// Render the set header as a JSON object. The timestamp is emitted as the
// §2.7 clock's seconds value rather than a formatted date: a set document is
// machine input, and a numeric instant cannot be misread by a reader in another
// locale. TimeSynchronized travels with it, so a consumer can tell a trustworthy
// instant from one stamped while the clock had lost its source.
METHOD M_Header : STRING(480)
VAR_INPUT
    Info : ST_ConfigSetInfo;
END_VAR
VAR
    nameText  : STRING(480);
    rootText  : STRING(480);
    modelText : STRING(480);
    line      : STRING(480);
    used      : INT;
    ok        : BOOL;
END_VAR
M_Header := '';
IF Info.SetName = '' THEN
    RETURN;
END_IF
nameText := _M_Escape(Text := Info.SetName, Ok => ok);
IF NOT ok THEN
    RETURN;
END_IF
rootText := _M_Escape(Text := Info.RootIdentity, Ok => ok);
IF NOT ok THEN
    RETURN;
END_IF
modelText := _M_Escape(Text := Info.ModelCode, Ok => ok);
IF NOT ok THEN
    RETURN;
END_IF
line := '';
used := 0;
ok := _M_PutText(Text := '{"set":"', Line := line, Used := used)
    AND_THEN _M_Put(pText := ADR(nameText), Line := line, Used := used)
    AND_THEN _M_PutText(Text := '","root":"', Line := line, Used := used)
    AND_THEN _M_Put(pText := ADR(rootText), Line := line, Used := used)
    AND_THEN _M_PutText(Text := '","schema":', Line := line, Used := used)
    AND_THEN _M_PutText(Text := UINT_TO_STRING(Info.SetSchema), Line := line, Used := used)
    AND_THEN _M_PutText(Text := ',"configRev":', Line := line, Used := used)
    AND_THEN _M_PutText(Text := UDINT_TO_STRING(Info.ConfigRev), Line := line, Used := used)
    AND_THEN _M_PutText(Text := ',"kind":', Line := line, Used := used)
    AND_THEN _M_PutText(Text := DINT_TO_STRING(TO_DINT(Info.Kind)), Line := line, Used := used)
    AND_THEN _M_PutText(Text := ',"model":"', Line := line, Used := used)
    AND_THEN _M_Put(pText := ADR(modelText), Line := line, Used := used)
    AND_THEN _M_PutText(Text := '","records":', Line := line, Used := used)
    AND_THEN _M_PutText(Text := INT_TO_STRING(Info.RecordCount), Line := line, Used := used)
    AND_THEN _M_PutText(Text := ',"created":', Line := line, Used := used)
    AND_THEN _M_PutText(Text := UDINT_TO_STRING(DT_TO_UDINT(Info.CreatedAt)), Line := line, Used := used)
    AND_THEN _M_PutText(Text := ',"clock":', Line := line, Used := used);
IF ok THEN
    IF Info.TimeSynchronized THEN
        ok := _M_PutText(Text := '1}', Line := line, Used := used);
    ELSE
        ok := _M_PutText(Text := '0}', Line := line, Used := used);
    END_IF
END_IF
IF ok THEN
    M_Header := line;
END_IF
END_METHOD

// Read one field out of a flat JSON object line. Deliberately NOT a general
// JSON parser: the accepted shape is exactly what M_Record and M_Header emit -
// a single object of scalar members, no nesting, no arrays. Anything else is
// refused rather than half-understood, which is the §14 rule for untrusted
// input applied to a format instead of to a value.
METHOD PRIVATE _M_Field : BOOL
VAR_INPUT
    Line : STRING(480);
    Name : STRING(32);
END_VAR
VAR_OUTPUT
    Value : STRING(255);
END_VAR
VAR
    pIn   : POINTER TO BYTE;
    pOut  : POINTER TO BYTE;
    buf   : STRING(255);
    token : STRING(40);
    pTok  : POINTER TO BYTE;
    tokLen : INT;
    found : INT;
    i     : INT;
    j     : INT;
    k     : INT;
    n     : INT;
    ch    : BYTE;
    quoted : BOOL;
END_VAR
_M_Field := FALSE;
Value := '';
buf := '';
token := CONCAT('"', CONCAT(Name, '":'));   // short: CONCAT is exact here
pIn := ADR(Line);
pTok := ADR(token);
n := _M_Length(pText := pIn);               // FIND/LEN would see only 255 of it
tokLen := TO_INT(LEN(token));
found := -1;
FOR i := 0 TO n - tokLen DO
    k := 0;
    WHILE (k < tokLen) AND_THEN (pIn[i + k] = pTok[k]) DO
        k := k + 1;
    END_WHILE
    IF k = tokLen THEN
        found := i;
        EXIT;
    END_IF
END_FOR
IF found < 0 THEN
    RETURN;                                // absent: the caller decides if that is fatal
END_IF
i := found + tokLen;                          // 0-based index of the first value byte
IF i >= n THEN
    RETURN;
END_IF
pOut := ADR(buf);
j := 0;
quoted := (pIn[i] = 16#22);
IF quoted THEN
    i := i + 1;
END_IF
WHILE i < n DO
    ch := pIn[i];
    IF quoted THEN
        IF ch = 16#22 THEN
            EXIT;                          // closing quote
        END_IF
        IF ch = 16#5C THEN
            i := i + 1;                    // unescape: the next byte is literal
            IF i >= n THEN
                RETURN;                    // trailing escape: malformed, refuse
            END_IF
            ch := pIn[i];
        END_IF
    ELSE
        IF (ch = 16#2C) OR (ch = 16#7D) THEN
            EXIT;                          // ',' or '}' ends a bare number
        END_IF
    END_IF
    IF j >= 254 THEN
        RETURN;                            // longer than any value we can store
    END_IF
    pOut[j] := ch;
    j := j + 1;
    i := i + 1;
END_WHILE
IF quoted AND (i >= n) THEN
    RETURN;                                // unterminated string: malformed
END_IF
pOut[j] := 0;
Value := buf;
_M_Field := TRUE;
END_METHOD

// Parse one record line back into a record. FALSE = the line is not a record
// line this build understands, and NOTHING in Record has been changed.
//
// This is untrusted input in the fullest sense - it may have been edited by
// hand, produced by another vendor's tool, or moved between machines - so it is
// parsed into a record and then still validated by the owning module's typed
// handler before any value changes (§5.6, §14). Getting a well-formed record
// out of here proves the SYNTAX, never the value.
METHOD M_ParseRecord : BOOL
VAR_INPUT
    Line : STRING(480);
END_VAR
VAR_IN_OUT
    Record : ST_ConfigRecord;
END_VAR
VAR
    scopeText : STRING(255);
    keyText   : STRING(255);
    valueText : STRING(255);
    revText   : STRING(255);
    kindText  : STRING(255);
    typeText  : STRING(255);
    revValue  : LREAL;
    kindValue : LREAL;
    typeValue : LREAL;
END_VAR
M_ParseRecord := FALSE;
IF NOT _M_Field(Line := Line, Name := 'key', Value => keyText) THEN
    RETURN;
END_IF
IF keyText = '' THEN
    RETURN;                                // a record without an identity is not one
END_IF
IF TO_INT(LEN(keyText)) > 160 THEN
    RETURN;                                // wider than the mutation identity: refuse
END_IF
IF NOT _M_Field(Line := Line, Name := 'scope', Value => scopeText) THEN
    RETURN;
END_IF
IF TO_INT(LEN(scopeText)) > 80 THEN
    RETURN;
END_IF
IF NOT _M_Field(Line := Line, Name := 'value', Value => valueText) THEN
    RETURN;
END_IF
IF TO_INT(LEN(valueText)) > 80 THEN
    RETURN;                                // wider than any registered text target
END_IF
IF NOT _M_Field(Line := Line, Name := 'rev', Value => revText) THEN
    RETURN;
END_IF
IF NOT _M_Field(Line := Line, Name := 'kind', Value => kindText) THEN
    RETURN;
END_IF
IF NOT _M_Field(Line := Line, Name := 'type', Value => typeText) THEN
    RETURN;
END_IF
IF NOT F_TryParseNumber(Text := revText, Value => revValue) THEN
    RETURN;
END_IF
IF (revValue < 1.0) OR (revValue > 4294967295.0) THEN
    RETURN;
END_IF
IF NOT F_TryParseNumber(Text := kindText, Value => kindValue) THEN
    RETURN;
END_IF
IF (kindValue < 0.0) OR (kindValue > DINT_TO_LREAL(TO_DINT(E_ConfigKind.LINE_CFG))) THEN
    RETURN;                                // outside E_ConfigKind: fail closed
END_IF
IF NOT F_TryParseNumber(Text := typeText, Value => typeValue) THEN
    RETURN;
END_IF
IF (typeValue < 0.0) OR (typeValue > 3.0) THEN
    RETURN;                                // outside E_ConfigValueType: fail closed
END_IF
// Every field is now known-good, so the record is filled in one go: a partially
// overwritten record handed back on a later failure would be worse than none.
Record.Scope := scopeText;
Record.WriteKey := keyText;
Record.ValueText := valueText;
Record.Revision := LREAL_TO_UDINT(revValue);
Record.Kind := LREAL_TO_DINT(kindValue);
Record.ValueType := LREAL_TO_DINT(typeValue);
M_ParseRecord := TRUE;
END_METHOD

// §3.8b — parse a set HEADER line. FALSE = not a header (no "set" member), or
// one this build cannot make sense of; Info is untouched either way.
//
// A header and a record are unambiguous by shape - a header carries "set" and a
// record carries "key", and neither carries the other - so a caller can offer a
// line to both and let the document tell it what the line is.
METHOD M_ParseHeader : BOOL
VAR_INPUT
    Line : STRING(480);
END_VAR
VAR_IN_OUT
    Info : ST_ConfigSetInfo;
END_VAR
VAR
    nameText  : STRING(255);
    rootText  : STRING(255);
    modelText : STRING(255);
    schemaText : STRING(255);
    revText   : STRING(255);
    kindText  : STRING(255);
    countText : STRING(255);
    createdText : STRING(255);
    clockText : STRING(255);
    schema    : LREAL;
    configRev : LREAL;
    kind      : LREAL;
    records   : LREAL;
    created   : LREAL;
    clock     : LREAL;
END_VAR
M_ParseHeader := FALSE;
IF NOT _M_Field(Line := Line, Name := 'set', Value => nameText) THEN
    RETURN;                                // not a header line
END_IF
IF nameText = '' THEN
    RETURN;
END_IF
IF TO_INT(LEN(nameText)) > 80 THEN
    RETURN;
END_IF
IF NOT _M_Field(Line := Line, Name := 'root', Value => rootText) THEN
    RETURN;
END_IF
IF TO_INT(LEN(rootText)) > 80 THEN
    RETURN;
END_IF
IF NOT _M_Field(Line := Line, Name := 'model', Value => modelText) THEN
    RETURN;
END_IF
IF TO_INT(LEN(modelText)) > 64 THEN
    RETURN;
END_IF
IF NOT _M_Field(Line := Line, Name := 'schema', Value => schemaText) THEN
    RETURN;
END_IF
IF NOT _M_Field(Line := Line, Name := 'configRev', Value => revText) THEN
    RETURN;
END_IF
IF NOT _M_Field(Line := Line, Name := 'kind', Value => kindText) THEN
    RETURN;
END_IF
IF NOT _M_Field(Line := Line, Name := 'records', Value => countText) THEN
    RETURN;
END_IF
IF NOT _M_Field(Line := Line, Name := 'created', Value => createdText) THEN
    RETURN;
END_IF
IF NOT _M_Field(Line := Line, Name := 'clock', Value => clockText) THEN
    RETURN;
END_IF
IF NOT F_TryParseNumber(Text := schemaText, Value => schema) THEN
    RETURN;
END_IF
IF (schema < 0.0) OR (schema > 65535.0) THEN
    RETURN;
END_IF
IF NOT F_TryParseNumber(Text := revText, Value => configRev) THEN
    RETURN;
END_IF
IF (configRev < 0.0) OR (configRev > 4294967295.0) THEN
    RETURN;
END_IF
IF NOT F_TryParseNumber(Text := kindText, Value => kind) THEN
    RETURN;
END_IF
IF (kind < 0.0) OR (kind > DINT_TO_LREAL(TO_DINT(E_ConfigKind.LINE_CFG))) THEN
    RETURN;                                // outside E_ConfigKind: fail closed
END_IF
IF NOT F_TryParseNumber(Text := countText, Value => records) THEN
    RETURN;
END_IF
IF (records < 0.0) OR (records > 32767.0) THEN
    RETURN;
END_IF
IF NOT F_TryParseNumber(Text := createdText, Value => created) THEN
    RETURN;
END_IF
IF (created < 0.0) OR (created > 4294967295.0) THEN
    RETURN;
END_IF
IF NOT F_TryParseNumber(Text := clockText, Value => clock) THEN
    RETURN;
END_IF
// Filled only once every field is known-good: a partially overwritten header
// handed back on a later failure would describe a set that does not exist.
Info.Used := TRUE;
Info.SetName := nameText;
Info.RootIdentity := rootText;
Info.ModelCode := modelText;
Info.SetSchema := LREAL_TO_UINT(schema);
Info.ConfigRev := LREAL_TO_UDINT(configRev);
Info.Kind := LREAL_TO_DINT(kind);
Info.RecordCount := LREAL_TO_INT(records);
Info.CreatedAt := UDINT_TO_DT(LREAL_TO_UDINT(created));
Info.TimeSynchronized := (clock <> 0.0);
M_ParseHeader := TRUE;
END_METHOD

END_FUNCTION_BLOCK

// ---- Platform/F_TryParseNumber.TcPOU
// Core §3.8b/§5.6 — parse a client-supplied decimal number, rejecting anything
// that is not one. The plain conversion cannot be used on its own: STRING_TO_LREAL
// answers 0 for '', 'abc' and '12kg' alike, so a configuration handler built on it
// accepts garbage as a valid zero and writes it. Every character is therefore
// checked before the conversion runs, and the caller learns whether the text WAS a
// number separately from what the number is.
FUNCTION F_TryParseNumber : BOOL
VAR_INPUT
    Text : STRING(255);
END_VAR
VAR_OUTPUT
    Value : LREAL;
END_VAR
VAR
    i      : INT;
    n      : INT;
    c      : BYTE;
    digits : INT;
    dots   : INT;
    pc     : POINTER TO BYTE;
END_VAR

F_TryParseNumber := FALSE;
Value := 0.0;
n := TO_INT(LEN(Text));
// 40 characters is far more than any finite decimal this contract carries, and
// bounds the scan (§5.6).
IF (n <= 0) OR (n > 40) THEN
    RETURN;
END_IF
pc := ADR(Text);
digits := 0;
dots := 0;
FOR i := 0 TO n - 1 DO
    c := pc[i];
    IF (c >= 48) AND (c <= 57) THEN         // '0'..'9'
        digits := digits + 1;
    ELSIF c = 46 THEN                       // '.'
        dots := dots + 1;
        IF dots > 1 THEN
            RETURN;
        END_IF
    ELSIF ((c = 43) OR (c = 45)) AND (i = 0) THEN
        ;                                   // leading '+'/'-' only
    ELSE
        RETURN;                             // whitespace included: no silent trim
    END_IF
END_FOR
IF digits = 0 THEN
    RETURN;                                 // '-', '.', '+.' are not numbers
END_IF
Value := STRING_TO_LREAL(Text);
F_TryParseNumber := TRUE;

END_FUNCTION

// ---- Connectivity/FB_RetainPersistMedium.TcPOU
// Core §3.8b - the RETENTIVE-MEMORY medium (E_ConfigStore.LOCAL_RETAIN): a
// bounded pool of documents in the controller's PERSISTENT area, made durable
// by the shipped FB_PersistentDataWriter after every write. For a station with
// no usable file system, or one whose project prefers retentive memory.
//
// Limits stated, not hidden:
//   * MAX_RETAIN_DOCUMENTS documents of up to MAX_PERSIST_DOC_BYTES each, all
//     reserved in the persistent budget (8 x 16 kB as shipped); a write that
//     finds no free slot fails and is reported.
//   * A document's CRC catches a damaged copy, but a persistent image TwinCAT
//     itself could not restore comes back as a first boot: this medium cannot
//     tell that loss from an empty machine. The file medium can.
//   * PERSISTENT data is restored by symbol, so the pool is symbol-readable over
//     ADS. It is excluded from OPC UA, but it is NOT confidential: a credential
//     store refuses this medium (M_Confidential = FALSE).
FUNCTION_BLOCK FB_RetainPersistMedium EXTENDS FB_PersistMediumBase
VAR_OUTPUT
    StorageError : UDINT;   // last error (0 = none)
END_VAR
VAR PERSISTENT
    {attribute 'OPC.UA.DA' := '0'}
    _schema : UINT;
    {attribute 'OPC.UA.DA' := '0'}
    _docs : ARRAY[1..PL_Fraktal.MAX_RETAIN_DOCUMENTS] OF ST_RetainDocument;
END_VAR
VAR
    _checked  : BOOL;
    _rejected : BOOL;      // an unrecognized pool was cleared: reads report Lost
    {attribute 'OPC.UA.DA' := '0'}
    _writer   : FB_PersistentDataWriter;
    _phase    : INT;
END_VAR
VAR CONSTANT
    POOL_SCHEMA : UINT := 1;
    NO_SPACE    : UDINT := 16#70A;  // ADSERR_DEVICE_NOMEMORY
    TOO_LARGE   : UDINT := 16#705;
END_VAR

// no cyclic body: every caller's M_Poll advances the medium

METHOD M_Kind : E_ConfigStore
M_Kind := E_ConfigStore.LOCAL_RETAIN;
END_METHOD

METHOD M_Confidential : BOOL
M_Confidential := FALSE;
END_METHOD

METHOD PROTECTED _M_Step : BOOL
VAR
    i    : INT;
    slot : INT;
    free : INT;
END_VAR
_M_Step := FALSE;
_M_Check();
IF _phase = 1 THEN              // a write waiting for the persistent image
    IF NOT _writer.M_Cyclic() THEN
        _qResult[_active].Ok := NOT _writer.M_Failed();
        IF _writer.M_Failed() THEN
            _qResult[_active].ErrorId := INVALID_REQUEST;
            StorageError := INVALID_REQUEST;
        ELSE
            StorageError := 0;
        END_IF
        _phase := 0;
        _M_Step := TRUE;
    END_IF
    RETURN;
END_IF
slot := 0;
free := 0;
FOR i := 1 TO PL_Fraktal.MAX_RETAIN_DOCUMENTS DO
    IF _docs[i].Key = _qKey[_active] THEN
        slot := i;
    ELSIF (_docs[i].Key = '') AND (free = 0) THEN
        free := i;
    END_IF
END_FOR
IF NOT _qWrite[_active] THEN
    _qResult[_active].Ok := TRUE;
    _qResult[_active].Lost := _rejected;
    IF slot > 0 THEN
        IF (_docs[slot].Length = 0) OR (_docs[slot].Length > PL_Fraktal.MAX_PERSIST_DOC_BYTES) THEN
            _qResult[_active].Lost := TRUE;
        ELSIF F_Crc32(pData := ADR(_docs[slot].Data), Size := _docs[slot].Length) <> _docs[slot].Crc THEN
            _qResult[_active].Lost := TRUE;
        ELSIF _docs[slot].Length > _qSize[_active] THEN
            _qResult[_active].Ok := FALSE;
            _qResult[_active].ErrorId := TOO_LARGE;
        ELSE
            MEMCPY(destAddr := _qData[_active], srcAddr := ADR(_docs[slot].Data),
                n := _docs[slot].Length);
            _qResult[_active].Found := TRUE;
            _qResult[_active].Length := _docs[slot].Length;
        END_IF
    END_IF
    _M_Step := TRUE;
    RETURN;
END_IF
// Write. A zero-length document frees the slot.
IF _qSize[_active] = 0 THEN
    IF slot > 0 THEN
        _docs[slot].Key := '';
        _docs[slot].Length := 0;
    END_IF
ELSE
    IF slot = 0 THEN
        slot := free;
    END_IF
    IF slot = 0 THEN
        _qResult[_active].ErrorId := NO_SPACE;
        StorageError := NO_SPACE;
        _M_Step := TRUE;
        RETURN;
    END_IF
    MEMCPY(destAddr := ADR(_docs[slot].Data), srcAddr := _qData[_active],
        n := _qSize[_active]);
    _docs[slot].Length := _qSize[_active];
    _docs[slot].Crc := F_Crc32(pData := ADR(_docs[slot].Data), Size := _qSize[_active]);
    _docs[slot].Generation := _docs[slot].Generation + 1;
    _docs[slot].Key := _qKey[_active];      // last: the slot is claimed once whole
END_IF
_writer.M_Request();
_phase := 1;
END_METHOD

// §3.8b - the pool is versioned like every retained image: 0 is a first boot,
// any other unrecognized version is a rejected pool, cleared and reported.
METHOD PRIVATE _M_Check
VAR
    i : INT;
END_VAR
IF _checked THEN
    RETURN;
END_IF
_checked := TRUE;
IF _schema = POOL_SCHEMA THEN
    RETURN;
END_IF
_rejected := _schema <> 0;
FOR i := 1 TO PL_Fraktal.MAX_RETAIN_DOCUMENTS DO
    _docs[i].Key := '';
    _docs[i].Length := 0;
END_FOR
_schema := POOL_SCHEMA;
END_METHOD

END_FUNCTION_BLOCK

// ---- Connectivity/FB_PersistentDataWriter.TcPOU
// Core §3.8b — the SHIPPED DEFAULT durability provider for E_ConfigStore
// .LOCAL_RETAIN: it makes the PLC's retentive image reach non-volatile storage
// on demand, so an accepted configuration write is DURABLE and not merely LIVE.
//
// Why this exists at all: on TwinCAT the persistent image is written by the
// runtime, normally at a controlled shutdown. Every configuration write since
// the last write is therefore lost to a power cut - the station silently
// reverts at its next restart, which is exactly the failure §3.8b replaces with
// a stated property. Requesting the write explicitly turns that hope into an
// operation with a latency, a completion and a failure mode the root publishes.
//
// The ADS port is read from the runtime's own _AppInfo rather than hard-coded:
// a station on port 852 must not silently persist port 851's image.
FUNCTION_BLOCK FB_PersistentDataWriter IMPLEMENTS I_ConfigPersistence
VAR
    _writer  : Tc2_Utilities.FB_WritePersistentData;
    _busy    : BOOL;      // a write is in flight
    _queued  : BOOL;      // a request arrived while one was in flight
    _failed  : BOOL;      // latched until the next SUCCESSFUL write
END_VAR

// Driven through M_Cyclic by the owning root; no standalone scan behaviour.
;

// A write already in flight cannot be told about a value accepted after it
// started, so a request arriving now is QUEUED rather than merged: the value
// gets its own write and PersistPending stays TRUE until that one finishes.
// Merging them is the bug that reports a value durable which was never written.
METHOD M_Request : BOOL
_queued := TRUE;                           // picked up by the next M_Cyclic
M_Request := TRUE;
END_METHOD

// Drive the ADS write. Returns TRUE while data is still not durable, which is
// what the root publishes as PersistPending.
METHOD M_Cyclic : BOOL
IF _busy THEN
    _writer(START := FALSE);
    IF NOT _writer.BUSY THEN
        _busy := FALSE;
        _failed := _writer.ERR;
    END_IF
ELSIF _queued THEN
    _queued := FALSE;
    _busy := TRUE;
    // SPDM_2PASS is Beckhoff's optimized two-pass mode: the boot image stays
    // consistent even if the write is interrupted, which is the only mode worth
    // using for data whose whole purpose is surviving an uncontrolled stop.
    _writer(NETID := '',
            PORT := TwinCAT_SystemInfoVarList._AppInfo.AdsPort,
            START := TRUE,
            TMOUT := T#10S,
            MODE := Tc2_Utilities.SPDM_2PASS);
    IF NOT _writer.BUSY THEN
        // Refused before it began (bad port, runtime not accepting): that is a
        // completed failure, not an operation still in progress.
        _busy := FALSE;
        _failed := TRUE;
    END_IF
END_IF
M_Cyclic := _busy OR _queued;
END_METHOD

METHOD M_Failed : BOOL
M_Failed := _failed;
END_METHOD

END_FUNCTION_BLOCK

// ---- BaseClasses/FB_SequenceBase.TcPOU
// Core §6.8 — THE provided step-chain base: an SFC/ST/LD sequence POU extends
// this and gets the step record, condition waits, run-style pacing, the child
// PLCopen drive, delays, and the shared transition result — without re-declaring
// host plumbing per chain. The derived chart's actions are the only writers of
// _retVal; every chart transition reads it; one shared exit action calls
// M_ClearTransition. Framework flow-control lives here ONCE (§6.8(a)); the
// application's command/wait/decision logic stays visible in each step action.
FUNCTION_BLOCK ABSTRACT FB_SequenceBase IMPLEMENTS I_Sequence
VAR_OUTPUT
    ActiveStep : INT;              // §6.5 mirror of the step record (chart-local view)
    Done : BOOL;                   // finite chains: TRUE at their finish step
END_VAR
VAR
    _step    : INT;                // §6.5 active step index (the ST `CASE _step OF` token)
    // Shared transition result (§6.10). ONE-SCAN signal: the active step's action
    // is its only writer, every chart transition reads it, and it is cleared before
    // the next scan's actions run - by M_Advance on commit in an ST chart, or by
    // M_BeginScan when the chart runtime owns the transition (SFC/LD/FBD).
    _retVal  : E_StepResult;
    // §6.12 — the same one-scan signal as _retVal, but one per CONCURRENT LEG.
    // A parallel divergence has several active steps at once, so a single shared
    // result cannot work: whichever leg wrote last would decide every leg's
    // transition. Index n belongs to leg n; the main line keeps _retVal, so a
    // chain with no parallel branch never touches this array.
    //
    // A leg's step action writes `_conRetVal[n] := E_StepResult.ADVANCE;` and its
    // transition reads `_conRetVal[n] = E_StepResult.ADVANCE`; the join reads every
    // leg plus the main line. Cleared with _retVal once per scan (M_BeginScan), and
    // per leg on that leg's step exit (M_ClearTransition) - never across legs,
    // which would let one leg's commit erase another's result mid-motion.
    _conRetVal  : ARRAY[1..PL_Fraktal.MAX_PARALLEL_BRANCHES] OF E_StepResult;
    _restart : BOOL;               // a step may request a chart restart (M_Run applies it)
    // Native chart restart, consumed by the initial step's mandatory M_Step.
    // SFC POUs enable Reset/use-inherited in their archive; ST/LD ignore it.
    {attribute 'OPC.UA.DA' := '0'}
    SFCReset : BOOL;
    {attribute 'OPC.UA.DA' := '0'}
    _host : I_SequenceHost;        // owning module's framework services (§6.7)
    _attached : BOOL;
    // §6.12 — every STEP-scoped latch is per CONCURRENT BRANCH, because two legs of
    // a parallel divergence are two active steps in the same POU at the same time.
    // Sharing one latch let leg A's issue consume leg B's, and let leg A's step exit
    // wipe leg B's transition result. Index 0 is the main line, which is what a chain
    // without any parallel branch uses throughout.
    _delay : ARRAY[0..PL_Fraktal.MAX_PARALLEL_BRANCHES] OF TON;
    _driveIssued : ARRAY[0..PL_Fraktal.MAX_PARALLEL_BRANCHES] OF BOOL;
    _subRunning : ARRAY[0..PL_Fraktal.MAX_PARALLEL_BRANCHES] OF BOOL;
    // Which leg the step action executing RIGHT NOW belongs to. Set by M_Step from
    // its `Branch` input, so it is always in step with the record just published,
    // and reset to _branchBase every scan - a chain that never names a leg is
    // therefore always on its own, which for a top-level chain is the main line.
    _branch : INT;
    // This chain's own leg index when the chain IS a leg (assigned by M_RunPar at
    // the fork). 0 for a top-level chain. It is what lets a leg written as its own
    // chain tag every one of its rows without naming a branch anywhere.
    _branchBase : INT;
    _lastStep : ARRAY[0..PL_Fraktal.MAX_PARALLEL_BRANCHES] OF INT;
    _stepSeen : ARRAY[0..PL_Fraktal.MAX_PARALLEL_BRANCHES] OF BOOL;
    _parStarted : ARRAY[1..PL_Fraktal.MAX_PARALLEL_BRANCHES] OF BOOL;
    _parLegs : INT;                // M_RunPar calls made this scan
    _parDone : INT;                // how many of them reported Done
    _errorRaised : BOOL;           // this chain raised the active fault (§6.9)
    _warnRaised : ARRAY[0..PL_Fraktal.MAX_PARALLEL_BRANCHES] OF BOOL;   // §6.9(e) one message per step visit
    _baseStepNo : INT;             // §6.5 step-record offset when run as a sub-chain
END_VAR

;

// §6.8 ST-skeleton progression: at the END of a `CASE _step OF` body, commit the
// step's shared transition result. On ADVANCE (or a declared JUMPn) go to the
// mapped next step and clear the step-scoped latches so the new step re-arms — the
// exact guarantee the SFC exit action gave, in one call. NONE stays put. The caller
// passes its successor map; an unmapped result holds the step (safe, visible).
METHOD M_Advance
VAR_INPUT
    OnAdvance : INT;               // next step for E_StepResult.ADVANCE
    // Jump targets default to "not used" so the common case reads
    // `M_Advance(OnAdvance := 100);` instead of repeating `OnJump1..3 := -1`.
    // Defaulted METHOD inputs need TwinCAT >= 3.1.4026, so on the legacy 4024
    // target (FRAKTAL_TC3_4024 defined) they are declared without defaults and
    // every argument is passed explicitly. See Params/PL_FraktalCompat.TcGVL.
    {IF defined (FRAKTAL_TC3_4024)}
    OnJump1   : INT;               // next step for JUMP1 (-1 = not used)
    OnJump2   : INT;               // next step for JUMP2 (-1 = not used)
    OnJump3   : INT;               // next step for JUMP3 (-1 = not used)
    {ELSE}
    OnJump1   : INT := -1;         // next step for JUMP1 (-1 = not used)
    OnJump2   : INT := -1;         // next step for JUMP2 (-1 = not used)
    OnJump3   : INT := -1;         // next step for JUMP3 (-1 = not used)
    {END_IF}
END_VAR
VAR
    target : INT;
END_VAR
target := -1;
CASE _retVal OF
    E_StepResult.ADVANCE: target := OnAdvance;
    E_StepResult.JUMP1:   target := OnJump1;
    E_StepResult.JUMP2:   target := OnJump2;
    E_StepResult.JUMP3:   target := OnJump3;
END_CASE
IF target >= 0 THEN
    _step := target;
    ActiveStep := target;
    M_ClearTransition();           // §6.10: a completed result never leaks into the next step
END_IF
END_METHOD

// §6.11 forward
METHOD M_AskDecision
VAR_INPUT
    Req : ST_DecisionRequest;
END_VAR
IF _host <> 0 THEN
    _host.M_SequenceAskDecision(Req := Req);
END_IF
END_METHOD

// bind the owner's host bridge; the derived Setup adds its typed child bindings.
METHOD M_Attach : BOOL
VAR_INPUT
    Host : I_SequenceHost;
END_VAR
_host := Host;
_attached := (Host <> 0);
IF _attached THEN
    // Announce this chain to its owner so the Unit base can run the
    // §6.10 per-scan result reset for it. The project writes nothing (O1).
    _host.M_SequenceRegister(Seq := THIS^);
END_IF
M_Attach := _attached;
END_METHOD

// §6.9(b) named plain-condition wait (forward to the host).
METHOD M_Await : BOOL
VAR_INPUT
    Idx : INT;
    Label : STRING(120);
    Ok : BOOL;
END_VAR
M_Await := FALSE;
IF _host <> 0 THEN
    M_Await := _host.M_SequenceAwait(Idx := Idx, Label := Label, Ok := Ok);
END_IF
END_METHOD

// Core §6.10 - scan-scoped reset of the shared transition result.
//
// `_retVal` is a ONE-SCAN signal: the active step's action writes it, the chart's
// transition reads it in the same scan, and it must not survive into the next.
// In an ST chart M_Advance is itself the transition, so it commits and clears in
// one call. In a chart language the RUNTIME evaluates transitions (SFC/LD/FBD),
// so nothing in the chart is positioned to clear afterwards - call this once per
// PLC cycle immediately BEFORE executing the chart. Clearing at the top of the
// scan is equivalent to clearing after the previous scan's transitions, and it
// forces every step action to re-assert its own result each scan, which is the
// property that makes a stale ADVANCE impossible.
//
// It deliberately clears ONLY the result. `_driveIssued` (M_TryIssue's one-shot)
// and `_delay` (M_Delay's timer) are STEP-scoped, not scan-scoped: resetting them
// every scan would re-issue a child command every cycle and stop any delay from
// ever elapsing. Those re-arm on step change, through M_ClearTransition.
METHOD M_BeginScan
VAR
	Idx : INT;
END_VAR
_retVal := E_StepResult.NONE;
FOR Idx := 1 TO PL_Fraktal.MAX_PARALLEL_BRANCHES DO
    _conRetVal[Idx] := E_StepResult.NONE;
END_FOR
// §6.12 the branch cursor is scan-scoped: a step action that does not declare a
// branch is on the main line (or on this chain's own leg when it IS a leg), so a
// chain with no parallel branch never mentions one.
_branch := _branchBase;
_parLegs := 0;
_parDone := 0;
END_METHOD

// Restart this chain as a sub-chain of a composite step: its step records are
// offset by the owning step number (§6.5) so the stall walk still reports one
// continuous chain. OnChainReset carries any application state.
METHOD M_ChainReset
VAR_INPUT
    BaseStepNo : INT;
    // §6.12 the leg index this chain runs as, assigned by the fork. 0 = not a leg.
    // Every step it records is tagged with it, so the project writes it once per
    // leg instead of once per step (§1.1 O1).
    Branch : INT;
END_VAR
_baseStepNo := BaseStepNo;
_branchBase := Branch;
M_ResetBase(FirstStep := 0);
OnChainReset();
SFCReset := TRUE; // request native graph reset after shared flow reset
END_METHOD

// §6.12 — the join of a parallel step: ADVANCE on the scan every leg run this
// scan has reported Done, NONE while any is still working. The counts are
// scan-scoped, so the join always reflects the legs the step actually ran -
// there is no leg list to register, and none to forget to update (§1.1 O1).
METHOD M_ParJoin : E_StepResult
M_ParJoin := E_StepResult.NONE;
IF (_parLegs > 0) AND (_parDone = _parLegs) THEN
    M_ParJoin := E_StepResult.ADVANCE;
END_IF
END_METHOD

// §6.12 — run one leg of a parallel step. THE portable form of a parallel
// divergence, and the only one available to an ST chain.
//
//     M_Step(StepNo := 500, StepName := 'project.step.bothPositions', ...);
//     M_RunPar(Chain := _positionA, BaseStepNo := 500, Branch := 1);
//     M_RunPar(Chain := _positionB, BaseStepNo := 600, Branch := 2);
//     _retVal := M_ParJoin();
//     M_Advance(OnAdvance := 999);
//
// Each leg is an ordinary FB_SequenceBase chain, so it brings its own step
// pointer, its own transition result and its own step-scoped latches - the
// collisions §6.12 has to manage inside one POU simply cannot arise (§1.1 O4:
// the model scales structurally rather than by decoration). Its steps are
// recorded under BaseStepNo and tagged with Branch, so the §3.13 flow chart
// groups them and the §6.9 walk still names one continuous chain.
//
// Returns TRUE on the scans this leg reports Done. The entry latch is
// step-scoped, so re-entering the fork step later restarts every leg.
METHOD M_RunPar : BOOL
VAR_INPUT
    Chain : REFERENCE TO FB_SequenceBase;
    BaseStepNo : INT;
    Branch : INT;
END_VAR
M_RunPar := FALSE;
IF NOT __ISVALIDREF(Chain) THEN
    RETURN;
END_IF
IF (Branch < 1) OR (Branch > PL_Fraktal.MAX_PARALLEL_BRANCHES) THEN
    M_Fault(Reason := E_Reason.UNSUPPORTED_COMMAND,
        DescriptionKey := 'std.error.parallelBranchOutOfRange');
    RETURN;                          // §5.6 no silent default
END_IF
IF NOT _parStarted[Branch] THEN
    Chain.M_ChainReset(BaseStepNo := BaseStepNo, Branch := Branch);
    _parStarted[Branch] := TRUE;
END_IF
Chain.M_ChainRun();
_parLegs := _parLegs + 1;
IF Chain.Done THEN
    _parDone := _parDone + 1;
    M_RunPar := TRUE;
END_IF
END_METHOD

// One scan of this chain. An ST chart overrides this with its
// `CASE _step OF` body; a chart-language POU leaves it alone because its own body
// IS the chart and the runtime executes it. Only a chain that is used as a
// composite step (M_RunSub) has to override it.
METHOD M_ChainRun
;
END_METHOD

METHOD M_ClearDecision
IF _host <> 0 THEN
    _host.M_SequenceClearDecision();
END_IF
END_METHOD

// the ONE shared STEP-EXIT action: a completed step's result never leaks into
// the next step, and the step-scoped helpers (delay, drive latch) re-arm.
// §6.12 — it re-arms THE CURRENT BRANCH only. Clearing every branch here is what
// made a parallel divergence misbehave: one leg committing a step wiped the other
// leg's transition result and its issue latch mid-motion.
// ST charts reach this through M_Advance on commit. A chart language whose
// engine owns the transition (SFC/LD/FBD) wires this as the step exit action,
// which the runtime executes AFTER the transition condition was evaluated -
// so the transition still sees the result the step action produced.
METHOD M_ClearTransition
VAR
	Idx : INT;
END_VAR
IF _branch = 0 THEN
    _retVal := E_StepResult.NONE;
    // A fork always sits on the main line of its own chain (§6.12), so leaving the
    // fork step is what re-arms its legs for a later re-entry.
    FOR Idx := 1 TO PL_Fraktal.MAX_PARALLEL_BRANCHES DO
        _parStarted[Idx] := FALSE;
    END_FOR
ELSE
    _conRetVal[_branch] := E_StepResult.NONE;
END_IF
_driveIssued[_branch] := FALSE;
_warnRaised[_branch] := FALSE;
_subRunning[_branch] := FALSE;
_delay[_branch](IN := FALSE);
END_METHOD

// §6.1 one-shot completion forward (finite chains)
METHOD M_Complete
IF _host <> 0 THEN
    _host.M_SequenceComplete();
END_IF
END_METHOD

METHOD M_CountGood
IF _host <> 0 THEN
    _host.M_SequenceCountGood();
END_IF
END_METHOD

// a declared process wait in ONE step (settle/dwell). The timer runs while the
// step is active and re-arms through the shared exit action.
METHOD M_Delay : E_StepResult
VAR_INPUT
    PT : TIME;
END_VAR
M_Delay := E_StepResult.NONE;
_delay[_branch](IN := TRUE, PT := PT);
IF _delay[_branch].Q THEN
    _delay[_branch](IN := FALSE);
    M_Delay := E_StepResult.ADVANCE;
END_IF
END_METHOD

// §8.11.1 cycle-complete marker forward; FALSE = stop granted (do not loop)
METHOD M_EndOfCycle : BOOL
M_EndOfCycle := FALSE;
IF _host <> 0 THEN
    M_EndOfCycle := _host.M_SequenceEndOfCycle();
END_IF
END_METHOD

// §6.9 first-out fault from a step (forward to the host).
METHOD M_Fault
VAR_INPUT
    Reason : E_Reason;
    DescriptionKey : STRING(255);
END_VAR
IF _host <> 0 THEN
    _host.M_SequenceFault(Reason := Reason, DescriptionKey := DescriptionKey);
END_IF
END_METHOD

// §3.4.2 run-style pacing gate (forward to the host).
METHOD M_Gate : BOOL
VAR_INPUT
    Steppable : BOOL;
END_VAR
M_Gate := FALSE;
IF _host <> 0 THEN
    M_Gate := _host.M_SequenceStepGate(Steppable := Steppable);
END_IF
END_METHOD

// §6.1 issue+await in ONE step: TRUE exactly once per step visit, when the
// run-style gate permits (§3.4.2). The action then sets the child's typed
// Command and raises Execute — visibly, in the step (§6.8). The child's Done
// releases the handshake and sets _retVal := ADVANCE; a child Error needs no
// step code — the owning Unit adopts it instantly via the §8.2 rollup.
// The latch re-arms through the shared exit action (M_ClearTransition).
METHOD M_TryIssue : BOOL
VAR_INPUT
    Steppable : BOOL;
END_VAR
M_TryIssue := FALSE;
IF _driveIssued[_branch] THEN
    RETURN;
END_IF
IF M_Gate(Steppable := Steppable) THEN
    _driveIssued[_branch] := TRUE;
    M_TryIssue := TRUE;
END_IF
END_METHOD

METHOD M_PartProcessed : BOOL
VAR_INPUT
    Verdict : E_Verdict;
    Reason : E_Reason;
END_VAR
M_PartProcessed := FALSE;
IF _host <> 0 THEN
    M_PartProcessed := _host.M_SequencePartProcessed(Verdict := Verdict, Reason := Reason);
END_IF
END_METHOD

// §3.16.3 forward (framework plumbing stays out of step actions).
METHOD M_PartReceived : BOOL
M_PartReceived := FALSE;
IF _host <> 0 THEN
    M_PartReceived := _host.M_SequencePartReceived();
END_IF
END_METHOD

METHOD M_PartRecord : BOOL
VAR_INPUT
    RecordName : STRING(64);
    Value : LREAL;
    Minimum : LREAL;
    Maximum : LREAL;
    Target : LREAL;
    EngUnit : STRING(16);
END_VAR
M_PartRecord := FALSE;
IF _host <> 0 THEN
    M_PartRecord := _host.M_SequencePartRecord(RecordName := RecordName,
        Value := Value, Minimum := Minimum, Maximum := Maximum, Target := Target,
        EngUnit := EngUnit);
END_IF
END_METHOD

METHOD M_PartStarted
IF _host <> 0 THEN
    _host.M_SequencePartStarted();
END_IF
END_METHOD

// §6.9/§8.8 — raise a message this step defines itself.
//
// For a condition the framework cannot see: a measured value out of band, a
// disagreement between two children, an application rule. LinkPath is the module
// the §3.13 chart should drill into ('' = this Unit).
//
// Severity and Category are a PROPOSAL, not the last word: adoption runs the §8.8
// rationalization, so a reason that is in the registry gets the registry's priority
// and category and these inputs are ignored. They survive for a project band code
// (10000+) the registry does not know - which is exactly where a custom message of
// a different level belongs.
METHOD M_RaiseCustom : BOOL
VAR_INPUT
    Reason         : E_Reason;
    DescriptionKey : STRING(255);
    Severity       : E_Severity;
    Category       : E_Category;
    LinkPath       : STRING(255);
END_VAR
VAR
    diag : ST_Diagnostic;
END_VAR
M_RaiseCustom := FALSE;
IF _host = 0 THEN
    RETURN;
END_IF
diag.ReasonCode  := Reason;
diag.Description := DescriptionKey;
diag.SourcePath  := LinkPath;
diag.Severity    := Severity;
diag.Category    := Category;
M_RaiseCustom := _host.M_SequenceRaise(Diag := diag, LinkPath := LinkPath);
_errorRaised := M_RaiseCustom;
END_METHOD

// §6.9 — adopt a child's first-out from inside conditional step logic.
//
// `Awaits` rolls a child fault up automatically, but only for a step that hands
// the child to the framework. A step that decides for itself - anything with an
// IF or CASE around the command - calls this instead, and gets the same result:
// the child's reason verbatim, the child's path as the §3.13 drill-down link,
// and the chain stopped until the error is cleared.
//
// Returns TRUE only when a fault was actually raised, so the usual shape is
//     IF M_RaiseFromChild(Source := _pressRam) THEN RETURN; END_IF
METHOD M_RaiseFromChild : BOOL
VAR_INPUT
    Source : I_Module;
END_VAR
M_RaiseFromChild := FALSE;
IF Source = 0 THEN
    RETURN;
END_IF
IF NOT Source.FaultActive THEN
    RETURN;                          // nothing to raise: safe to call every scan
END_IF
IF _host = 0 THEN
    RETURN;
END_IF
M_RaiseFromChild := _host.M_SequenceRaise(Diag := Source.GetFaultSummary(),
    LinkPath := Source.Name);
_errorRaised := M_RaiseFromChild;
END_METHOD

// §6.9(e) — a custom message that informs and lets the chain carry on.
//
// For designed behaviour with a consequence worth recording: an operator
// releasing a two-hand control mid-motion, a retry, a value drifting inside its
// band. It is NOT the error path - the chain is not stopped, no fault is
// adopted, and the step keeps whatever recovery it already routes to.
//
// Raised at most ONCE per visit to a step, however many scans the step runs and
// however many times this is called (§1.1 O1: a project shall never have to
// remember an edge latch for correctness). Committing the step re-arms it.
//
// Severity/Category are the caller's for a project band code; a reason in the
// §8.8 registry is rationalized to the registry's values like any other.
METHOD M_RaiseWarning : BOOL
VAR_INPUT
    Reason         : E_Reason;
    DescriptionKey : STRING(255);
    Severity       : E_Severity;
    Category       : E_Category;
END_VAR
VAR
    diag : ST_Diagnostic;
END_VAR
M_RaiseWarning := FALSE;
IF _warnRaised[_branch] OR (_host = 0) THEN
    RETURN;                          // already said once for this visit
END_IF
diag.ReasonCode  := Reason;
diag.Description := DescriptionKey;
diag.Severity    := Severity;
diag.Category    := Category;
M_RaiseWarning := _host.M_SequenceWarn(Diag := diag);
_warnRaised[_branch] := M_RaiseWarning;
END_METHOD

// §6.9(e) — publish a child's failure WITHOUT adopting it.
//
// The counterpart of M_RaiseFromChild, for a step that already owns the
// recovery: the child's first-out reaches the alarm ring and the §3.13 chart
// (marked on this step, click-through to the child), but nothing faults and the
// chain keeps the branch it was going to take anyway. Press AUTO N200 is the
// case: the ram not reaching is handled by an operator confirmation and a scrap,
// so stopping there would replace a designed recovery with a hard fault - while
// saying nothing left the failure invisible on the Unit.
//
// Reported once per visit to the step, so calling it every scan is correct.
METHOD M_ReportFromChild : BOOL
VAR_INPUT
    Source : I_Module;
END_VAR
M_ReportFromChild := FALSE;
IF _warnRaised[_branch] OR (_host = 0) OR (Source = 0) THEN
    RETURN;
END_IF
IF NOT Source.FaultActive THEN
    RETURN;                          // nothing to report: safe every scan
END_IF
M_ReportFromChild := _host.M_SequenceWarn(Diag := Source.GetFaultSummary());
_warnRaised[_branch] := M_ReportFromChild;
END_METHOD

// clear the base flow state to the first step. The derived M_Reset calls this.
METHOD M_ResetBase
VAR_INPUT
    // Defaults to 0 (N000), the conventional first step, so a derived M_Reset
    // reads `M_ResetBase();`. Legacy 4024 has no defaulted method inputs, so
    // there the argument is required — see Params/PL_FraktalCompat.TcGVL.
    {IF defined (FRAKTAL_TC3_4024)}
    FirstStep : INT;               // the chain's initial step number (N000 = 0)
    {ELSE}
    FirstStep : INT := 0;          // the chain's initial step number (N000 = 0)
    {END_IF}
END_VAR
VAR
    Idx : INT;
END_VAR
_step := FirstStep;
ActiveStep := FirstStep;
Done := FALSE;
_restart := FALSE;
SFCReset := FALSE;
// §6.12 a reset re-arms EVERY branch, not just the one that happened to run last.
FOR Idx := 0 TO PL_Fraktal.MAX_PARALLEL_BRANCHES DO
    _stepSeen[Idx] := FALSE;
    _lastStep[Idx] := -1;
    _branch := Idx;
    M_ClearTransition();
END_FOR
_branch := _branchBase;
_parLegs := 0;
_parDone := 0;
END_METHOD

// §6.8 I_Sequence - start over at N000 with the chain's own state cleared. The
// owning Unit calls this for every attached chain on first scan, mode change and
// both abort paths, and a project calls it (through _M_RestartSequences) where
// its own restart-or-resume policy says so. A chain puts the state it owns in
// OnChainReset and writes no reset method of its own (§1.1 O1).
METHOD M_Restart
M_ResetBase(FirstStep := 0);
OnChainReset();
SFCReset := TRUE; // request native graph reset after shared flow reset
END_METHOD

// §6.9 — the owning Unit left ERROR. The chain's _step was never touched, so it
// resumes exactly where it stopped; re-arming the step-scoped latches here is
// what makes it RE-EVALUATE the command rather than resume mid-handshake with a
// spent M_TryIssue one-shot and a half-run delay.
METHOD M_ResumeAfterError
IF NOT _errorRaised THEN
    RETURN;
END_IF
_errorRaised := FALSE;
M_ClearTransition();
END_METHOD

// §6.8 run another chain as ONE composite step. Returns NONE while the
// sub-chain works and ADVANCE on the scan it finishes, so a step action reads:
//
//     _retVal := M_RunSub(Chain := _loadPosition, BaseStepNo := 240);
//
// The entry latch is step-scoped and re-arms through M_ClearTransition, so a
// chain re-entered later restarts correctly. The sub-chain inherits the leg of
// the step that runs it (§6.12), so a composite step inside a parallel branch
// publishes its sub-steps under that leg without saying so. Hand-written, this was eight lines
// per composite step and one forgotten latch reset left a chain that never ran
// again (§1.1 O1: the framework owns repeated flow control, not the project).
METHOD M_RunSub : E_StepResult
VAR_INPUT
    Chain : REFERENCE TO FB_SequenceBase;
    BaseStepNo : INT;
END_VAR
M_RunSub := E_StepResult.NONE;
IF NOT __ISVALIDREF(Chain) THEN
    RETURN;
END_IF
IF NOT _subRunning[_branch] THEN
    // §6.12 — the sub-chain runs INSIDE this step, so it belongs to whatever leg
    // this step is on. _branch is already correct (M_Step set it from the step
    // record), so there is nothing for the project to state and nothing that can
    // drift out of step with the record - the same reason Branch is an input of
    // M_Step rather than a call beside it (§1.1 O1).
    Chain.M_ChainReset(BaseStepNo := BaseStepNo, Branch := _branch);
    _subRunning[_branch] := TRUE;
END_IF
Chain.M_ChainRun();
IF Chain.Done THEN
    _subRunning[_branch] := FALSE;
    M_RunSub := E_StepResult.ADVANCE;
END_IF
END_METHOD

// §6.5 step record + the chart-local ActiveStep mirror, one call.
METHOD M_Step
VAR_INPUT
    StepNo : INT;
    StepName : STRING(120);
    Awaits : I_Module;
    AwaitingLabel : STRING(120);
    TimeClass : E_TimeClass;
    ExpectedTime : TIME;
    // §6.12 — the concurrent leg this step belongs to, which a step on the main
    // line never mentions. Folding it into the step record rather than a separate
    // call is what makes it impossible to declare a leg without recording a step,
    // or to record a step under the wrong leg because the declaration was
    // forgotten (§1.1 O1: the framework owns the bookkeeping, not the project).
    // 0 means "this chain's own leg", which is the main line for a top-level chain
    // and the index the fork assigned for a chain running as a leg (M_RunPar) -
    // so a leg written as its own chain never mentions a branch either.
    {IF defined (FRAKTAL_TC3_4024)}
    Branch : INT;
    {ELSE}
    Branch : INT := 0;
    {END_IF}
END_VAR
// §6.12 — select the leg first: everything below, and everything the step action
// does after this call (M_TryIssue, M_Delay, M_RunSub, the §6.9(e) message latch)
// is scoped to it. An out-of-range index faults rather than quietly landing on the
// main line (§5.6 - no silent default).
IF Branch < 0 OR Branch > PL_Fraktal.MAX_PARALLEL_BRANCHES THEN
    M_Fault(Reason := E_Reason.UNSUPPORTED_COMMAND,
        DescriptionKey := 'std.error.parallelBranchOutOfRange');
    RETURN;
END_IF
// SFCReset executes the initial action; its mandatory M_Step consumes the pulse.
// Every chart gets the same restart behavior without a project reset call.
SFCReset := FALSE;
IF Branch > 0 THEN
    _branch := Branch;
ELSE
    _branch := _branchBase;
END_IF
// A chart language never calls M_ClearTransition: its engine owns the transition,
// so there is no commit point to hang it on. The step record is the one call every
// step of every language makes, so the re-arm belongs here - a new step number on
// this leg re-arms that leg's issue latch, delay and message. Without it
// M_TryIssue fired once per chart RUN instead of once per step.
IF (NOT _stepSeen[_branch]) OR (_lastStep[_branch] <> StepNo) THEN
    _lastStep[_branch] := StepNo;
    _stepSeen[_branch] := TRUE;
    M_ClearTransition();
END_IF
ActiveStep := StepNo;
IF _host <> 0 THEN
    _host.M_SequenceSetStep(StepNo := StepNo, StepName := StepName, Awaits := Awaits,
        AwaitingLabel := AwaitingLabel, TimeClass := TimeClass, ExpectedTime := ExpectedTime,
        Branch := _branch);
END_IF
END_METHOD

// §3.4/§8.11 — accept the stop between cycles (forward to the host).
METHOD M_StopNow
IF _host <> 0 THEN
    _host.M_SequenceStopNow();
END_IF
END_METHOD

// §3.4 — poll at the between-cycles wait step (forward to the host).
METHOD M_StopPending : BOOL
M_StopPending := FALSE;
IF _host <> 0 THEN
    M_StopPending := _host.M_SequenceStopPending();
END_IF
END_METHOD

METHOD M_TakeDecision : INT
M_TakeDecision := 0;
IF _host <> 0 THEN
    M_TakeDecision := _host.M_SequenceTakeDecision();
END_IF
END_METHOD

// §3.14 hook: clear application-owned chain state on restart. Empty by default
// so a chain that has none writes nothing.
METHOD PROTECTED OnChainReset
;
END_METHOD

END_FUNCTION_BLOCK

// ---- BaseClasses/FB_UnitBase.TcPOU
// Core §2.2 lifecycle family, top tier: modes + cascade (§3.4/§3.7), Start/Stop
// mapped onto the §6.1 run command (§6 intro), the step chain (_M_SetStep/_M_Await,
// §6.5/§6.9(b)), the stall walk as a PENDING reason with instant rollup on an
// awaited module's Error (§6.9/§8.2), the §8.11.4 profiler wired in, and
// Starved/Blocked derived from the step's time class (§8.11.4(f)/§8.11.3).
// A Unit type overrides _M_Dispatch (its mode chain) + _M_Supports (+ §3.14 hooks).
FUNCTION_BLOCK ABSTRACT FB_UnitBase EXTENDS FB_CompositeModuleBase IMPLEMENTS I_Unit, I_SequenceHost
VAR_INPUT
    DecisionAnswer : INT;              // §6.11: chosen option index (0 = none yet)
    ReqControlOn   : BOOL;             // §9.8 HMI/data request; edge-consumed and access-gated
    ReqControlOff  : BOOL;
    HmiRequest     : ST_HmiRequest;     // §3.10/§14: arguments first, Sequence last
    {attribute 'OPC.UA.DA' := '0'}
    ControlDomain  : ST_ControlDomainStatus; // §9.8: optional shared cell/cage arrangement
END_VAR
VAR_OUTPUT
    Starved : BOOL;                    // §8.11.3 — derived from CurrentStep.TimeClass
    Blocked : BOOL;
    Domain  : ST_ControlDomainStatus;  // §9.8 read-only publication of the assigned domain
    ControlOnRequest  : BOOL;          // one-scan request to the owning domain coordinator
    ControlOffRequest : BOOL;
END_VAR
VAR_OUTPUT
    Profiler    : FB_CycleProfiler;    // §8.11.4 — HMI chart source
    CurrentStep : ST_StepRecord;       // §6.5 — feeds §6.9 walk AND the profiler
    // §3.13 sequence flow chart. Discovered from _M_SetStep, so a chain author
    // writes nothing; SequenceStepCount is the published length (§8.4 bounded).
    SequenceSteps : ARRAY[1..PL_Fraktal.MAX_SEQUENCE_STEPS] OF ST_SequenceStep;
    // §3.10.2 — the static half of each row: discovered once, never changes, so it
    // stays OFF the cyclic tree and is served through the config manifest under the
    // SAME browse paths as the live half (M_AppendConfig below).
    {attribute 'OPC.UA.DA' := '0'}
    SequenceStepDef : ARRAY[1..PL_Fraktal.MAX_SEQUENCE_STEPS] OF ST_SequenceStepDef;
    // §3.13 — which row each concurrent leg is running. Indexed by branch (0 = the
    // main line), so it is ~10 entries however long the chain is, and cheap enough
    // to stay in the cyclic read: the chart is right the moment its tab opens.
    ActiveSteps : ARRAY[0..PL_Fraktal.MAX_PARALLEL_BRANCHES] OF ST_SequenceCursor;
    // §6.9 — the errors and messages currently attached to rows. Sparse, so a small
    // table instead of 633 bytes reserved on every row for the usually-empty case.
    SequenceAnnotations : ARRAY[1..PL_Fraktal.MAX_SEQUENCE_ANNOTATIONS] OF ST_SequenceAnnotation;
    SequenceAnnotationCount : INT;
    SequenceStepCount : INT;
    CurrentStepElapsed : TIME;         // how long the active step has been running
    CurrentStepTimedOut : BOOL;        // active step outran its guard (§6.9 stall)

    Pending     : ST_Diagnostic;       // live stall reason (Low) — NOT a fault (§6.9)
    Decision    : ST_DecisionRequest;  // §6.11 active request ('' Prompt = none)
    {attribute 'OPC.UA.DA' := '0'}
    StallTime   : TIME := T#30S;       // guard when the step declares no ExpectedTime
    Model       : ST_ModelId;          // §3.1b active model identity (published for HMI/MES/trace)
    // §3.10.2 — static catalogs served via the QUERY_CONFIG manifest, not cyclically
    {attribute 'OPC.UA.DA' := '0'}
    ModelCapacity : INT;
    {attribute 'OPC.UA.DA' := '0'}
    Features : ST_ConfigFeatures := (ExportCurrentConfig := TRUE);
    {attribute 'OPC.UA.DA' := '0'}
    AvailableModelCount : INT;         // §3.8 optional discoverable model/recipe catalog
    {attribute 'OPC.UA.DA' := '0'}
    AvailableModels : ARRAY[1..PL_Fraktal.MAX_RECIPES] OF ST_ModelId;
    Part        : ST_PartContext;      // §3.16.1 live part context (Present=FALSE, Uid='' = none)
    AlarmLog    : FB_AlarmLog;         // §8.3 — active list + closed ring + Blocking
    HostEvents  : FB_HostEventPublisher; // §11.6 fixed, bounded L3/MES projection
    Access      : FB_AccessManager;    // §7.7 — per-root session/policy (default: fully open)
    GoodCount   : UDINT;               // §8.11.2 — cycle verdict counters
    NokCount    : UDINT;
    ReworkCount : UDINT;
    NokReason   : E_Reason;            // §8.11.2 — last NOK's first-out attribution
    MachineState : E_MachineState;     // §8.11.3 — classified every scan (OEE/PackML/host)
    History     : ARRAY[1..PL_Fraktal.MAX_DIAG_RING] OF ST_Diagnostic;  // §6.9(a) ring (newest at HistoryHead)
    HistoryHead : INT;
    {attribute 'OPC.UA.DA' := '0'}
    ModePolicy  : ARRAY[0..PL_Fraktal.MODE_COUNT-1] OF ST_ModePolicy;    // §3.4.1 per-mode switch policy (station cfg; manifest-served)
    RunStyle    : E_RunStyle;          // §3.4.2 active run style (HMI-selectable; CONTINUOUS default)
    Oee         : ST_Oee;              // §8.5.1 accumulators + snapshot (published)
    // §8.5.2 - shifts, when a line is referenced (SetLine). 0 = no shift accounting.
    CurrentShift          : INT;
    ShiftStartedAt        : DT;
    ShiftProductionTarget : UDINT;
    ShiftHistory          : ARRAY[1..PL_Fraktal.MAX_SHIFT_HISTORY] OF ST_ShiftRecordV3; // newest first; released V1 type remains unchanged
    ShiftHistoryCount     : INT;
    ShiftHistoryTruncated : BOOL;
    OeeTrend    : ARRAY[1..PL_Fraktal.MAX_OEE_SAMPLES] OF ST_OeeSample; // §8.5.1 ring
    OeeTrendHead: INT;                 // newest sample index (0 = none yet)
    HmiResponse : ST_HmiResponse;
    ConfigRev   : UDINT;                // §3.10.2 manifest revision — HMI refetches on change
    // §3.8b — is this station's configuration actually SAFE? Transport
    // acknowledgement and Accepted mean a value is LIVE; this says whether it is
    // DURABLE, whether anything was lost at the last restart, and what the last
    // set operation did. Published cyclically because the answer changes without
    // anybody asking, and because it has to be visible BEFORE the restart that
    // would otherwise reveal it.
    ConfigPersist : ST_ConfigPersistStatus;
    // §3.8b — the store's set listing, refreshed on a LIST_CONFIG_SETS request.
    // Published, and read ON DEMAND: a client target-reads it when a set dialog
    // opens, never in its cyclic snapshot (§1.1 O4). It was marked DA := '0' until
    // 2026-09-27, which made the listing and the export lines unreachable over OPC
    // UA altogether - a client could request them and never read the answer.
    ConfigSets : ARRAY[1..PL_Fraktal.MAX_CONFIG_SETS] OF ST_ConfigSetInfo;
    ConfigSetCount : INT;
    // §3.8b — one line of a set's JSON document, served by EXPORT_CONFIG_SET.
    // Line 0 is the header and 1..RecordCount are the records, so a client pulls
    // a movable document a line at a time without a full buffer in the PLC —
    // the same paging discipline QUERY_CONFIG already uses.
    ConfigSetDocument : STRING(480);
    ConfigSetDocumentLine : INT;
    ConfigSetDocumentLines : INT;
    ModeActivePublished : E_Mode;       // properties are not OPC UA-visible
    RunningPublished : BOOL;
    StopPendingPublished : BOOL;
    SupportedModesPublished : ARRAY[0..PL_Fraktal.MODE_COUNT-1] OF BOOL;
    SupportedRunStylesPublished : ARRAY[0..2] OF BOOL;
    SystemHealth : ST_SystemHealthStatus; // §2.7/§8.12 live, trendable health
    SignalTower  : ST_SignalTowerOut;     // §8.13 single reusable mapping
END_VAR
VAR PERSISTENT
    // §3.8a station-config backing for the manifest-served ModePolicy output.
    // Version 0/unrecognized initializes safe defaults exactly once.
    _modePolicyVersion : UINT;
    _modePolicyStored : ARRAY[0..PL_Fraktal.MODE_COUNT-1] OF ST_ModePolicy;
END_VAR
VAR
    _fTrig    : R_TRIG;
    _mode     : E_Mode;
    _modeReq  : E_Mode;
    _modePend : BOOL;
    _modeExitFirst : BOOL;
    _stopReq  : BOOL;
    {attribute 'OPC.UA.DA' := '0'}
    _awaits   : I_Module;              // module the current step awaits (0 = none)
    _faultEvt : INT;                   // open ERROR event slot in AlarmLog (0 = none)
    _tStall   : TON;
    _seqIndex : INT;                   // row recorded LAST, i.e. the step action running now
    _stepSinceMs : DWORD;              // monotonic start of the main-line step
    // §6.12 — per-row clock and liveness. With a parallel step several rows are
    // active at once, so one cursor is no longer enough to say what is running or
    // for how long. Bounded exactly like the row table itself (§1.1 O10).
    // Per-LEG, not per row: a leg has one active step, so the per-scan sweep is ~10
    // iterations instead of up to MAX_SEQUENCE_STEPS.
    _branchSinceMs : ARRAY[0..PL_Fraktal.MAX_PARALLEL_BRANCHES] OF DWORD;
    _branchTouched : ARRAY[0..PL_Fraktal.MAX_PARALLEL_BRANCHES] OF BOOL;
    _tDecision: TON;                   // §6.11 monotonic active-decision timeout
    _decisionConflictLogged : BOOL;    // one audit record per conflicting request
    _decisionResolutionLogged : BOOL;  // operator/timeout resolution logged once
    _stepReq  : BOOL;                  // §3.4.2 pending single-step request (edge-consumed)
    _holdRun  : BOOL;                  // §3.4.2 HOLD_TO_RUN input held (NON-SAFETY, §9)
    _stepArm  : R_TRIG;
    _errClr   : R_TRIG;                // §6.9 the ERROR state ended
    _oeeLast  : TIME;                  // §8.5.1 last accumulation stamp
    _oeeSampMs: UDINT;                 // ms since last trend sample
    // §8.5.2 shift accounting
    {attribute 'OPC.UA.DA' := '0'}
    _pLine : POINTER TO FB_LineData;
    // §3.8a - model data: the provider and key of this root's own recipe record,
    // and the buffer a model-scoped request loads another model's record into.
    {attribute 'OPC.UA.DA' := '0'}
    _modelProvider : I_RecipeProvider;
    {attribute 'OPC.UA.DA' := '0'}
    _modelCatalog : I_RecipeCatalog;
    {attribute 'OPC.UA.DA' := '0'}
    _snapshot : FB_ConfigSnapshot;
    {attribute 'OPC.UA.DA' := '0'}
    _loadSnapshot : FB_ConfigSnapshot;
    _exportToken : STRING(160);
    _exportSession : UDINT;
    _exportNext : INT;
    _exportName : STRING(80);
    _modelCatalogSeen : INT := -1;
    _modelKey : STRING(80);
    _viewModelCode : STRING(64);
    {attribute 'OPC.UA.DA' := '0'}
    _modelBuf : ARRAY[1..PL_Fraktal.MAX_MODEL_DATA_BYTES] OF BYTE;
    _lineHost : BOOL;                  // §3.8e this root ticks the line it references
    _lineRevSeen : UDINT;              // §3.8e line revision last reflected in ConfigRev
    _shiftEnd : DT;
    _shiftLastNow : DT;
    _shiftCalendarRev : UDINT;
    _oeeGoodBase : UDINT;
    _oeeNokBase : UDINT;
    _shiftInit : BOOL;
    _shiftSync : BOOL;
    _shiftManualReset : BOOL;
    _hmiLastSequence : UDINT;
    {attribute 'OPC.UA.DA' := '0'}
    _configPager : FB_ConfigPager;     // §3.10.2 QUERY_CONFIG window writer
    // §3.8b — the parameter-set store. Absent (the shipped default for a Unit
    // nobody wired one into) means save/load/list are simply not offered, which
    // is published as StorePresent = FALSE rather than failing at the first
    // request an operator makes.
    {attribute 'OPC.UA.DA' := '0'}
    _configStore : I_ConfigStore;
    // §3.8b durability. _persistWriter is the shipped LOCAL_RETAIN default and
    // is used unless a deployment injects something else, so a conforming
    // station persists its parametrization with no file system, no network and
    // no configuration — and with no line of project code either (§1.1 O1).
    {attribute 'OPC.UA.DA' := '0'}
    _persistWriter : FB_PersistentDataWriter;
    {attribute 'OPC.UA.DA' := '0'}
    _persistence : I_ConfigPersistence;
    _persistSinceMs : DWORD;           // monotonic ms the current window started at
    _persistEvt : INT;                 // open PersistFailed event slot (0 = none)
    _restoreEvt : INT;                 // open restore-loss event slot (0 = none)
    {attribute 'OPC.UA.DA' := '0'}
    _setJson : FB_ConfigSetJson;       // §3.8b text projection (export/import)
    // §3.8b - the project's persistence MEDIUM (SetPersistMedium): this root's live
    // station, line and model data kept as documents on it and restored at start.
    // Absent (the shipped default) = the native PERSISTENT data alone.
    {attribute 'OPC.UA.DA' := '0'}
    _medium : I_PersistMedium;
    {attribute 'OPC.UA.DA' := '0'}
    _liveDoc : FB_ConfigSetDocument;
    // A store that writes its sets out itself (FB_MediumConfigStore): found on the
    // injected store by __QUERYINTERFACE and driven beside _persistence.
    {attribute 'OPC.UA.DA' := '0'}
    _storePersistence : I_ConfigPersistence;
    _livePhase : INT;
    _liveItem : INT;                   // 1 station, 2 line, 3.. model n = item - 2
    _liveArmed : BOOL;                 // OnInit ran: the capability walk is complete
    _liveRestored : BOOL;
    _liveDirty : BOOL;                 // an accepted change is not yet in the documents
    _liveFailed : BOOL;                // the last pass did not write every document
    _liveModels : BOOL;                // model data is kept per model (_M_LiveModelsKept)
    _liveModelSlots : INT;             // highest model document known on the medium
    _liveRetry : TON;
    _importOpen : BOOL;                // an IMPORT_CONFIG_SET save is in progress
    // §3.8b - a set line arriving in pieces (IMPORT_CONFIG_SET, IntValue = 1).
    // A request carries 255 characters and a line may hold 480, so the HMI
    // splits it; the pieces are joined here, and nowhere else.
    {attribute 'OPC.UA.DA' := '0'}
    _importPart : STRING(480);
    // §7.6.1a hold-to-run. The request is LATCHED and re-asserted every scan,
    // because a mailbox delivers one request per sequence and the axis expects
    // to be asked every scan it should keep moving. The latch is what makes
    // that work over a transport; the deadline is what keeps it safe, since a
    // client that stops refreshing - closed, crashed, unplugged - lets the hold
    // expire instead of leaving the machine moving.
    _heldPath  : STRING(255);
    _heldValue : DINT;
    _heldActive : BOOL;
    _heldSinceMs : DWORD;
    // §3.13 - the flow chart changed and the manifest revision owes it a bump.
    // Held until the growth settles, so one burst of row discovery costs one
    // refetch instead of one per row (PL_Fraktal.CHART_REV_SETTLE_MS).
    _chartDirty : BOOL;
    _chartTouchedMs : DWORD;
    {attribute 'OPC.UA.DA' := '0'}
    _carrier  : I_PartCarrier;         // §3.16.2 injected part carrier (0 = traceability off)
    {attribute 'OPC.UA.DA' := '0'}
    _healthPublisher : FB_SystemHealthPublisher;
    {attribute 'OPC.UA.DA' := '0'}
    _healthInput : ST_SystemHealthInput;
    {attribute 'OPC.UA.DA' := '0'}
    _healthParCfg : ST_SystemHealthParCfg;
    _healthConfigured : BOOL;
    {attribute 'OPC.UA.DA' := '0'}
    _towerMapper : FB_SignalTower;
    {attribute 'OPC.UA.DA' := '0'}
    _towerParCfg : ST_SignalTowerParCfg;
    _lampTestRequest : BOOL;
    {attribute 'OPC.UA.DA' := '0'}
    _sequences : ARRAY[1..PL_Fraktal.MAX_SEQUENCES] OF I_Sequence;
    _sequenceCount : INT;
    // §7.5 commissioning/engineering gate register, injected by the composition
    // root. Absent (the shipped default) = a production image: no gate is
    // annunciated and ForceChannel refuses every request (fail closed).
    {attribute 'OPC.UA.DA' := '0'}
    _engineering : REFERENCE TO FB_EngineeringMode;
    // §7.5.2 open standing event per registered gate (0 = none open yet)
    _engineeringEvt : ARRAY[1..PL_Fraktal.MAX_ENGINEERING_GATES] OF INT;
END_VAR
VAR CONSTANT
    // §3.8b — layout version of the retained ModePolicy image. Bump it when a
    // member is added to ST_ModePolicy or the array is resized; the retained
    // image is then rejected and annunciated instead of read by field position.
    MODE_POLICY_SCHEMA : UINT := 1;
    // §3.8b — schema version stamped into every set this root produces, so a set
    // document that outlives the build that wrote it can be recognized rather
    // than guessed at (§13).
    CONFIG_SET_SCHEMA : UINT := 1;
    // §3.8b - a live-document pass that failed is tried again this often.
    LIVE_RETRY : TIME := T#10S;
    // §3.8b - a live document the medium could not read is asked for again this
    // often; until it answers, nothing is restored, written or started.
    LIVE_READ_RETRY : TIME := T#2S;
END_VAR

Cyclic();

// Core §7.8 helper — append one non-interlock reason (bounds-checked).
METHOD PROTECTED _M_AddReason
VAR_IN_OUT
    Report : ST_ReleaseReport;
END_VAR
VAR_INPUT
    Text : STRING(255);
    Reason : E_Reason;
    Kind : E_ReleaseKind;
END_VAR
IF Report.Count >= PL_Fraktal.MAX_RELEASE_REASONS THEN
    RETURN;
END_IF
Report.Count := Report.Count + 1;
Report.Reasons[Report.Count].Description := Text;
Report.Reasons[Report.Count].ReasonCode  := Reason;
Report.Reasons[Report.Count].SourcePath  := _name;
Report.Reasons[Report.Count].Kind        := Kind;
Report.Reasons[Report.Count].Bypassable  := FALSE;
END_METHOD

// Core §7.8 — concrete Units override to append the active mode's immediate
// entry/frontier records via PermIntlk.AppendFailed(SourcePath, Report). Future step waits
// stay in CurrentStep/Pending and are not blanket Start conditions. Base: nothing.
METHOD PROTECTED _M_AppendInterlocks
VAR_IN_OUT
    Report : ST_ReleaseReport;
END_VAR
;
END_METHOD

// Core §7.8 — target-aware hook for the MANUAL release rollup: a concrete Unit
// overrides to append the §7.6 Release<Function> conditions of the SPECIFIC target
// module. Base delegates to the Unit-level hook (non-breaking default).
METHOD PROTECTED _M_AppendManualInterlocks
VAR_INPUT
    TargetPath : STRING(255);
    Value : DINT;
END_VAR
VAR_IN_OUT
    Report : ST_ReleaseReport;
END_VAR
_M_AppendInterlocks(Report := Report);
END_METHOD

// §6.11 option-aware release seam. The base validates session, active prompt and
// option identity; a concrete Unit appends the ordinary process conditions that a
// "continue"-style option must satisfy. Safety and child interlocks still remain
// authoritative at their owning modules.
METHOD PROTECTED _M_AppendDecisionInterlocks
VAR_INPUT
    Option : INT;
END_VAR
VAR_IN_OUT
    Report : ST_ReleaseReport;
END_VAR
;
END_METHOD

// §6.11 — publish a typed decision request (single active slot)
METHOD PROTECTED _M_AskDecision
VAR_INPUT
    Req : ST_DecisionRequest;
END_VAR
VAR
    candidate : ST_DecisionRequest;
END_VAR
candidate := Req;
IF candidate.SourcePath = '' THEN
    candidate.SourcePath := _name;
END_IF
// A sequence presents the same request every scan while its step waits. That is
// idempotent. A different producer never overwrites the visible active request.
IF Decision.Prompt <> '' THEN
    IF _M_DecisionMatches(Req := candidate) THEN
        RETURN;
    END_IF
    IF NOT _decisionConflictLogged THEN
        _M_LogDecision(EventKey := 'std.audit.decisionOverlapRejected',
            SourcePath := candidate.SourcePath, Option := 0);
        _decisionConflictLogged := TRUE;
    END_IF
    RETURN;
END_IF
IF NOT _M_ValidateDecision(Req := candidate) THEN
    _M_LogDecision(EventKey := 'std.audit.decisionInvalidRejected',
        SourcePath := candidate.SourcePath, Option := candidate.Default);
    _M_Fault(E_Reason.UNSUPPORTED_COMMAND, 'std.error.invalidDecisionRequest');
    RETURN;
END_IF
Decision := candidate;
DecisionAnswer := 0;
_decisionConflictLogged := FALSE;
_decisionResolutionLogged := FALSE;
_tDecision(IN := FALSE);
_M_LogDecision(EventKey := 'std.audit.decisionRequested',
    SourcePath := Decision.SourcePath, Option := 0);
END_METHOD

// Clear the complete public slot and all private latches atomically.
METHOD PRIVATE _M_ClearDecisionState
VAR
    i : INT;
END_VAR
_tDecision(IN := FALSE);
DecisionAnswer := 0;
Decision.Prompt := '';
Decision.Default := 0;
Decision.Timeout := T#0S;
Decision.SourcePath := '';
FOR i := 1 TO PL_Fraktal.MAX_OPTIONS DO
    Decision.Options[i] := '';
END_FOR
_decisionConflictLogged := FALSE;
_decisionResolutionLogged := FALSE;
END_METHOD

// §6.11 one-slot resolver. Operator input wins if it is accepted in the same scan
// the timeout expires; _M_HandleHmiRequest runs immediately before this method.
METHOD PRIVATE _M_DecisionCyclic
IF _exec <> E_ExecState.BUSY THEN
    IF Decision.Prompt <> '' THEN
        _M_LogDecision(EventKey := 'std.audit.decisionWithdrawn',
            SourcePath := Decision.SourcePath, Option := 0);
        _M_ClearDecisionState();
    ELSE
        _tDecision(IN := FALSE);
    END_IF
    RETURN;
END_IF
IF Decision.Prompt = '' THEN
    _tDecision(IN := FALSE);
    RETURN;
END_IF
IF DecisionAnswer <> 0 THEN
    _tDecision(IN := FALSE);
    IF (DecisionAnswer < 1) OR (DecisionAnswer > PL_Fraktal.MAX_OPTIONS) THEN
        _M_LogDecision(EventKey := 'std.audit.decisionAnswerRejected',
            SourcePath := Decision.SourcePath, Option := DecisionAnswer);
        DecisionAnswer := 0;
        RETURN;
    END_IF
    IF Decision.Options[DecisionAnswer] = '' THEN
        _M_LogDecision(EventKey := 'std.audit.decisionAnswerRejected',
            SourcePath := Decision.SourcePath, Option := DecisionAnswer);
        DecisionAnswer := 0;
        RETURN;
    END_IF
    IF NOT _decisionResolutionLogged THEN
        _M_LogDecision(EventKey := 'std.audit.decisionOperatorResolved',
            SourcePath := Decision.SourcePath, Option := DecisionAnswer);
        _decisionResolutionLogged := TRUE;
    END_IF
    RETURN;
END_IF
IF Decision.Timeout <= T#0S THEN
    _tDecision(IN := FALSE);
    RETURN;
END_IF
_tDecision(IN := TRUE, PT := Decision.Timeout);
IF _tDecision.Q THEN
    DecisionAnswer := Decision.Default;             // validated when accepted
    _tDecision(IN := FALSE);
    _M_LogDecision(EventKey := 'std.audit.decisionTimeoutResolved',
        SourcePath := Decision.SourcePath, Option := DecisionAnswer);
    _decisionResolutionLogged := TRUE;
END_IF
END_METHOD

// Full value comparison makes repeated presentation idempotent while treating a
// changed option/default/timeout as a different request that must not overwrite.
METHOD PRIVATE _M_DecisionMatches : BOOL
VAR_INPUT
    Req : ST_DecisionRequest;
END_VAR
VAR
    i : INT;
END_VAR
_M_DecisionMatches := FALSE;
IF (Decision.Prompt <> Req.Prompt)
OR (Decision.Default <> Req.Default)
OR (Decision.Timeout <> Req.Timeout)
OR (Decision.SourcePath <> Req.SourcePath) THEN
    RETURN;
END_IF
FOR i := 1 TO PL_Fraktal.MAX_OPTIONS DO
    IF Decision.Options[i] <> Req.Options[i] THEN
        RETURN;
    END_IF
END_FOR
_M_DecisionMatches := TRUE;
END_METHOD

// Domain audit: request, rejection and resolution are closed MESSAGE events.
METHOD PRIVATE _M_LogDecision
VAR_INPUT
    EventKey : STRING(160);
    SourcePath : STRING(255);
    Option : INT;
END_VAR
VAR
    slot : INT;
    textValue : STRING(255);
    sourceValue : STRING(255);
END_VAR
textValue := EventKey;
IF Option <> 0 THEN
    textValue := CONCAT(textValue, ' option=');
    textValue := CONCAT(textValue, TO_STRING(Option));
END_IF
sourceValue := SourcePath;
IF sourceValue = '' THEN
    sourceValue := _name;
END_IF
slot := AlarmLog.Raise(Reason := E_Reason.NONE, Text := textValue,
    Source := sourceValue, Severity := E_Severity.LOW,
    Category := E_Category.PROCESS, ResetClass := E_ResetClass.AUTO_RESET);
IF slot > 0 THEN
    AlarmLog.Gone(Slot := slot);
END_IF
END_METHOD

// A finite timeout requires a real safe default. An indefinite request may omit
// Default, but every published request still needs at least one selectable option.
METHOD PRIVATE _M_ValidateDecision : BOOL
VAR_INPUT
    Req : ST_DecisionRequest;
END_VAR
VAR
    i : INT;
    hasOption : BOOL;
END_VAR
_M_ValidateDecision := FALSE;
IF (Req.Prompt = '') OR (Req.Timeout < T#0S) THEN
    RETURN;
END_IF
hasOption := FALSE;
FOR i := 1 TO PL_Fraktal.MAX_OPTIONS DO
    IF Req.Options[i] <> '' THEN
        hasOption := TRUE;
    END_IF
END_FOR
IF NOT hasOption THEN
    RETURN;
END_IF
IF (Req.Timeout > T#0S) OR (Req.Default <> 0) THEN
    IF (Req.Default < 1) OR (Req.Default > PL_Fraktal.MAX_OPTIONS) THEN
        RETURN;
    END_IF
    IF Req.Options[Req.Default] = '' THEN
        RETURN;
    END_IF
END_IF
_M_ValidateDecision := TRUE;
END_METHOD

// §6.9(b) — named plain-condition wait; returns the condition so steps read naturally
METHOD PROTECTED _M_Await : BOOL
VAR_INPUT
    Idx   : INT;
    Label : STRING(120);
    Ok    : BOOL;
END_VAR
IF (Idx >= 1) AND (Idx <= PL_Fraktal.MAX_STEP_CONDS) THEN
    CurrentStep.Conds[Idx].Label := Label;
    CurrentStep.Conds[Idx].Ok    := Ok;
END_IF
_M_Await := Ok;
END_METHOD

// §3.7 — offer the mode to child Units; a child may reject (graceful)
METHOD PROTECTED _M_CascadeMode
VAR_INPUT
    Mode : E_Mode;
END_VAR
VAR
    i  : INT;
    iu : I_Unit;
END_VAR
FOR i := 1 TO _nChild DO
    IF _children[i] <> 0 THEN
        IF __QUERYINTERFACE(_children[i], iu) THEN   // [TC3] capability query — TC3 §3.2
            iu.SetMode(Mode);
        END_IF
    END_IF
END_FOR
END_METHOD

METHOD PROTECTED _M_ClearPending
Pending.ReasonCode  := E_Reason.NONE;
Pending.Description := '';
Pending.TimeSynchronized := FALSE;
END_METHOD

// §14.3 security audit for accepted remote mutations. Operational methods may
// additionally emit their domain event (manual action, OEE reset, shelving); this
// record supplies the remote request kind and authenticated user without secrets.
METHOD PROTECTED _M_AuditHmiAccepted
VAR_INPUT
    Kind : E_HmiRequestKind;
    TargetPath : STRING(255);
    Accepted : BOOL;
END_VAR
VAR
    auditable : BOOL;
    auditSlot : INT;
    textValue : STRING(255);
    sourcePath : STRING(255);
END_VAR
IF NOT Accepted THEN
    RETURN;
END_IF
CASE Kind OF
    E_HmiRequestKind.SET_MODE, E_HmiRequestKind.SET_MODEL,
    E_HmiRequestKind.START, E_HmiRequestKind.STOP,
    E_HmiRequestKind.CONTROL_ON, E_HmiRequestKind.CONTROL_OFF,
    E_HmiRequestKind.OPERATOR_RESET, E_HmiRequestKind.DECISION_ANSWER,
    E_HmiRequestKind.MANUAL_COMMAND, E_HmiRequestKind.SET_RUN_STYLE,
    E_HmiRequestKind.STEP_REQUEST, E_HmiRequestKind.SET_HOLD_RUN,
    E_HmiRequestKind.RESET_OEE, E_HmiRequestKind.WRITE_CONFIG,
    E_HmiRequestKind.SHELVE_ALARM, E_HmiRequestKind.UNSHELVE_ALARM,
    E_HmiRequestKind.FORCE_CHANNEL, E_HmiRequestKind.SET_ACCESS_LEVEL,
    E_HmiRequestKind.SET_SESSION_TIMEOUT, E_HmiRequestKind.LAMP_TEST,
    E_HmiRequestKind.CAPTURE_CONFIG, E_HmiRequestKind.SAVE_CONFIG_SET,
    E_HmiRequestKind.LOAD_CONFIG_SET, E_HmiRequestKind.ACK_CONFIG_RESTORE,
    E_HmiRequestKind.IMPORT_CONFIG_SET, E_HmiRequestKind.DELETE_CONFIG_SET,
    E_HmiRequestKind.SET_CLASS_LEVEL, E_HmiRequestKind.CREATE_MODEL:
        auditable := TRUE;
ELSE
    auditable := FALSE;
END_CASE
IF NOT auditable THEN
    RETURN;
END_IF
Access.RecordActivity();
textValue := CONCAT('std.audit.hmiAccepted kind=', TO_STRING(TO_DINT(Kind)));
textValue := CONCAT(textValue, ' user=');
textValue := CONCAT(textValue, Access.CurrentUser);
// §3.8b — a set operation is audited WITH the set name and record count: "the
// operator loaded a set" is not an audit record anyone can act on later.
IF (Kind = E_HmiRequestKind.SAVE_CONFIG_SET)
OR (Kind = E_HmiRequestKind.LOAD_CONFIG_SET)
OR (Kind = E_HmiRequestKind.DELETE_CONFIG_SET) THEN
    textValue := CONCAT(textValue, ' set=');
    textValue := CONCAT(textValue, ConfigPersist.LastSetName);
    textValue := CONCAT(textValue, ' records=');
    textValue := CONCAT(textValue, INT_TO_STRING(ConfigPersist.LastSetRecords));
END_IF
sourcePath := TargetPath;
IF sourcePath = '' THEN
    sourcePath := _name;
END_IF
auditSlot := AlarmLog.Raise(Reason := E_Reason.NONE, Text := textValue,
    Source := sourcePath, Severity := E_Severity.LOW, Category := E_Category.SYSTEM,
    ResetClass := E_ResetClass.AUTO_RESET);
IF auditSlot > 0 THEN AlarmLog.Gone(Slot := auditSlot); END_IF
END_METHOD

// Module paths are qualified dotted Fraktal identities (§4.8). A request routed
// through this root may target the root itself or one descendant, never a peer.
METHOD PRIVATE _M_OwnsModulePath : BOOL
VAR_INPUT
    Path : STRING(255);
END_VAR
VAR
    prefix : STRING(255);
END_VAR
prefix := CONCAT(_name, '.');
_M_OwnsModulePath := (Path = _name) OR (FIND(Path, prefix) = 1);
END_METHOD

// call at the finish step (§8.11.1): publishes the profile; FALSE = stop granted
METHOD PROTECTED _M_EndOfCycle : BOOL
Profiler.CycleComplete();
IF _stopReq THEN
    _stopReq := FALSE;
    Execute := FALSE;
    _M_Complete();
    _M_EndOfCycle := FALSE;
ELSE
    _M_EndOfCycle := TRUE;
END_IF
END_METHOD

// §3.10/§14 — consume one committed OPC UA request exactly once.
METHOD PROTECTED _M_HandleHmiRequest
VAR
    modelId  : ST_ModelId;
    modeReq  : E_Mode;
    styleReq : E_RunStyle;
    gateReq  : E_GatedAction;
    levelReq : E_AccessLevel;
    alarmSlot : INT;
    policyValueValid : BOOL;
    configKindReq : E_ConfigKind;
END_VAR
IF HmiRequest.Sequence = _hmiLastSequence THEN
    RETURN;
ELSE
    _hmiLastSequence := HmiRequest.Sequence;
END_IF

HmiResponse.Accepted := FALSE;
HmiResponse.Diagnostic := '';
HmiResponse.Report.Count := 0;
HmiResponse.Report.Released := FALSE;
// A held line piece belongs to the very next import request. Anything else in
// between means the line was abandoned, so it is dropped rather than glued to
// whatever arrives later.
IF HmiRequest.Kind <> E_HmiRequestKind.IMPORT_CONFIG_SET THEN
    _importPart := '';
END_IF

IF (HmiRequest.Kind <> E_HmiRequestKind.EXPORT_CONFIG_SET)
AND (HmiRequest.Kind <> E_HmiRequestKind.EXPORT_CURRENT_CONFIG) THEN
    _exportNext := 0;
END_IF
CASE HmiRequest.Kind OF
    E_HmiRequestKind.LOGIN:
        HmiResponse.Accepted := Access.RequestLogin(User := HmiRequest.User, Secret := HmiRequest.Secret);
    E_HmiRequestKind.LOGOUT:
        HmiResponse.Accepted := Access.RequestLogout();
    E_HmiRequestKind.SET_MODE:
        IF (HmiRequest.IntValue >= 0) AND (HmiRequest.IntValue < PL_Fraktal.MODE_COUNT) THEN
            modeReq := HmiRequest.IntValue;
            HmiResponse.Accepted := SetMode(Mode := modeReq);
        ELSE
            HmiResponse.Diagnostic := 'std.error.unsupportedModeRequest';
        END_IF
    E_HmiRequestKind.SET_MODEL:
        modelId.ModelCode := HmiRequest.TextValue;
        HmiResponse.Accepted := SetModel(Id := modelId);
    E_HmiRequestKind.START:
        HmiResponse.Accepted := Start();
    E_HmiRequestKind.STOP:
        HmiResponse.Accepted := Stop();
    E_HmiRequestKind.CONTROL_ON:
        HmiResponse.Accepted := RequestControlPower(ControlOn := TRUE);
    E_HmiRequestKind.CONTROL_OFF:
        HmiResponse.Accepted := RequestControlPower(ControlOn := FALSE);
    E_HmiRequestKind.OPERATOR_RESET:
        HmiResponse.Accepted := OperatorReset();
    E_HmiRequestKind.DECISION_ANSWER:
        HmiResponse.Accepted := SubmitDecision(Option := TO_INT(HmiRequest.IntValue),
            Report := HmiResponse.Report);
    E_HmiRequestKind.MANUAL_COMMAND:
        HmiResponse.Accepted := ManualCommandTo(TargetPath := HmiRequest.TargetPath, Value := HmiRequest.IntValue);
    E_HmiRequestKind.MANUAL_HELD:
        HmiResponse.Accepted := ManualHeldTo(TargetPath := HmiRequest.TargetPath,
            Value := HmiRequest.IntValue, Held := HmiRequest.BoolValue);
    E_HmiRequestKind.SET_RUN_STYLE:
        IF (HmiRequest.IntValue >= 0) AND (HmiRequest.IntValue <= 2) THEN
            styleReq := HmiRequest.IntValue;
            HmiResponse.Accepted := SetRunStyle(Style := styleReq);
        ELSE
            HmiResponse.Diagnostic := 'std.error.unsupportedRunStyleRequest';
        END_IF
    E_HmiRequestKind.STEP_REQUEST:
        HmiResponse.Accepted := StepRequest();
    E_HmiRequestKind.SET_HOLD_RUN:
        HmiResponse.Accepted := SetHoldRun(Held := HmiRequest.BoolValue);
    E_HmiRequestKind.RELEASE_START:
        ReleaseReportStart(Report := HmiResponse.Report);
        HmiResponse.Accepted := TRUE;
    E_HmiRequestKind.RELEASE_MANUAL:
        ReleaseReportManual(TargetPath := HmiRequest.TargetPath, Value := HmiRequest.IntValue,
            Report := HmiResponse.Report);
        HmiResponse.Accepted := TRUE;
    E_HmiRequestKind.RELEASE_ACTION:
        IF (HmiRequest.IntValue >= 0)
        AND (HmiRequest.IntValue <= TO_DINT(E_GatedAction.CONFIG_SET)) THEN
            gateReq := HmiRequest.IntValue;
            ReleaseReportAction(Gate := gateReq, Report := HmiResponse.Report);
            HmiResponse.Accepted := TRUE;
        ELSE
            HmiResponse.Diagnostic := 'std.error.unsupportedGatedActionRequest';
        END_IF
    E_HmiRequestKind.RESET_OEE:
        HmiResponse.Accepted := ResetOee();
    E_HmiRequestKind.WRITE_CONFIG:
        // §3.8a - DurationMs names the model a model-data write is for
        // (0 = the active model, n = AvailableModels[n]); other values ignore it.
        HmiResponse.Accepted := WriteModelConfig(ModelIndex := HmiRequest.DurationMs,
            TargetPath := HmiRequest.TargetPath, WriteKey := HmiRequest.NameValue,
            Revision := HmiRequest.IntValue, TextValue := HmiRequest.TextValue);
    E_HmiRequestKind.SHELVE_ALARM:
        alarmSlot := AlarmLog.FindActiveSlot(SourcePath := HmiRequest.TargetPath,
            Description := HmiRequest.TextValue);
        IF alarmSlot > 0 THEN
            HmiResponse.Accepted := ShelveAlarm(Slot := alarmSlot,
                DurationS := HmiRequest.DurationMs / 1000);
        ELSE
            HmiResponse.Diagnostic := 'std.error.alarmIdentityNotUnique';
        END_IF
    E_HmiRequestKind.UNSHELVE_ALARM:
        alarmSlot := AlarmLog.FindActiveSlot(SourcePath := HmiRequest.TargetPath,
            Description := HmiRequest.TextValue);
        IF alarmSlot > 0 THEN
            HmiResponse.Accepted := UnshelveAlarm(Slot := alarmSlot);
        ELSE
            HmiResponse.Diagnostic := 'std.error.alarmIdentityNotUnique';
        END_IF
    E_HmiRequestKind.FORCE_CHANNEL:
        HmiResponse.Accepted := ForceChannel(ChannelPath := HmiRequest.TargetPath,
            Force := HmiRequest.BoolValue, BoolText := HmiRequest.TextValue,
            AnalogText := HmiRequest.NameValue);
    E_HmiRequestKind.QUERY_CONFIG:
        // §3.10.2 — serve one manifest page: re-walk the deterministic export
        // enumeration, storing only the requested window (no full buffer).
        // §3.8d: no blanket DATA_READ refusal any more - a class may be readable
        // below it. Each entry is served with or without its value by its level.
        _configPager.M_SetAccess(pAccess := ADR(Access));
        // §3.8a - DurationMs names the model whose model-data values to serve.
        IF NOT _configPager.M_Setup(Target := ADR(HmiResponse.ConfigPage),
            PageIndex := TO_INT(HmiRequest.IntValue), Revision := ConfigRev) THEN
            HmiResponse.Diagnostic := 'std.error.hmiRequestRejected';
        ELSIF M_AppendModelConfig(Pager := _configPager,
                ModelIndex := HmiRequest.DurationMs) THEN
            _configPager.M_Finish();
            HmiResponse.Accepted := TRUE;
        ELSE
            HmiResponse.Diagnostic := 'std.error.modelNotAvailable';
        END_IF
    E_HmiRequestKind.SET_ACCESS_LEVEL:
        policyValueValid := TRUE;
        IF HmiRequest.TextValue = '0' THEN
            levelReq := E_AccessLevel.NONE;
        ELSIF HmiRequest.TextValue = '1' THEN
            levelReq := E_AccessLevel.OPERATOR;
        ELSIF HmiRequest.TextValue = '2' THEN
            levelReq := E_AccessLevel.TECHNICIAN;
        ELSIF HmiRequest.TextValue = '3' THEN
            levelReq := E_AccessLevel.ENGINEER;
        ELSIF HmiRequest.TextValue = '4' THEN
            levelReq := E_AccessLevel.ADMIN;
        ELSE
            policyValueValid := FALSE;
        END_IF
        IF policyValueValid
        AND (HmiRequest.IntValue >= 0)
        AND (HmiRequest.IntValue <= TO_DINT(E_GatedAction.CONFIG_SET)) THEN
            gateReq := HmiRequest.IntValue;
            HmiResponse.Accepted := SetAccessLevel(Gate := gateReq, Level := levelReq);
        ELSE
            HmiResponse.Diagnostic := 'std.error.accessPolicyValueInvalid';
        END_IF
    E_HmiRequestKind.SET_SESSION_TIMEOUT:
        HmiResponse.Accepted := SetSessionTimeout(TimeoutMs := HmiRequest.DurationMs);
    E_HmiRequestKind.LAMP_TEST:
        HmiResponse.Accepted := RequestLampTest();
    E_HmiRequestKind.CAPTURE_CONFIG:
        // §3.8c(a) — a capture is routed through the SAME acknowledged mailbox as
        // the typed write it replaces, with the same arguments minus the value:
        // the number comes from the machine, not from the client.
        HmiResponse.Accepted := CaptureConfig(TargetPath := HmiRequest.TargetPath,
            WriteKey := HmiRequest.NameValue, Revision := HmiRequest.IntValue);
    E_HmiRequestKind.SAVE_CONFIG_SET:
        IF (HmiRequest.IntValue >= 0)
        AND (HmiRequest.IntValue <= TO_DINT(E_ConfigKind.LINE_CFG)) THEN
            configKindReq := HmiRequest.IntValue;
            HmiResponse.Accepted := SaveConfigSet(SetName := HmiRequest.TextValue,
                Kind := configKindReq);
        ELSE
            HmiResponse.Diagnostic := 'std.error.configSetKindInvalid';
        END_IF
    E_HmiRequestKind.LOAD_CONFIG_SET:
        HmiResponse.Accepted := LoadConfigSet(SetName := HmiRequest.TextValue);
        IF NOT HmiResponse.Accepted THEN
            HmiResponse.Diagnostic := 'std.error.configSetRejected';
        END_IF
    E_HmiRequestKind.LIST_CONFIG_SETS:
        HmiResponse.Accepted := ListConfigSets();
    E_HmiRequestKind.ACK_CONFIG_RESTORE:
        HmiResponse.Accepted := AcknowledgeConfigRestore();
        IF NOT HmiResponse.Accepted THEN
            HmiResponse.Diagnostic := 'std.error.configRestoreAckRefused';
        END_IF
    E_HmiRequestKind.EXPORT_CONFIG_SET:
        IF HmiRequest.NameValue <> '' THEN
            HmiResponse.Accepted := _M_ExportSnapshotLine(SetName := HmiRequest.TextValue,
                Line := TO_INT(HmiRequest.IntValue), Token := HmiRequest.NameValue);
        ELSE
            _exportNext := 0;
            HmiResponse.Accepted := ExportConfigSetLine(SetName := HmiRequest.TextValue,
                Line := TO_INT(HmiRequest.IntValue));
        END_IF
    E_HmiRequestKind.IMPORT_CONFIG_SET:
        HmiResponse.Accepted := ImportConfigSetPiece(Piece := HmiRequest.TextValue,
            More := HmiRequest.IntValue = 1, Commit := HmiRequest.BoolValue);
        IF NOT HmiResponse.Accepted THEN
            HmiResponse.Diagnostic := 'std.error.configSetLineRejected';
        END_IF
    E_HmiRequestKind.SET_CLASS_LEVEL:
        HmiResponse.Accepted := SetDataClassLevel(ClassId := HmiRequest.NameValue,
            Level := HmiRequest.IntValue, ForWrite := HmiRequest.BoolValue);
        IF NOT HmiResponse.Accepted THEN
            HmiResponse.Diagnostic := 'std.error.accessPolicyValueInvalid';
        END_IF
    E_HmiRequestKind.DELETE_CONFIG_SET:
        HmiResponse.Accepted := DeleteConfigSet(SetName := HmiRequest.TextValue);
        IF NOT HmiResponse.Accepted THEN
            HmiResponse.Diagnostic := 'std.error.configSetDeleteRefused';
        END_IF
    E_HmiRequestKind.CREATE_MODEL:
        IF HmiRequest.IntValue >= 0 THEN
            HmiResponse.Accepted := CreateModel(ModelCode := HmiRequest.NameValue,
                SourceIndex := TO_UDINT(HmiRequest.IntValue), FromSet := HmiRequest.BoolValue,
                SetName := HmiRequest.TextValue);
        END_IF
    E_HmiRequestKind.EXPORT_CURRENT_CONFIG:
        IF (HmiRequest.IntValue >= 0) AND (HmiRequest.IntValue <= TO_DINT(E_ConfigKind.LINE_CFG)) THEN
            configKindReq := HmiRequest.IntValue;
            HmiResponse.Accepted := ExportCurrentConfig(SetName := HmiRequest.TextValue,
                Kind := configKindReq, ModelIndex := HmiRequest.DurationMs,
                Token := HmiRequest.NameValue);
        END_IF
    E_HmiRequestKind.NONE:
        HmiResponse.Diagnostic := 'std.error.emptyHmiRequest';
ELSE
    HmiResponse.Diagnostic := 'std.error.unsupportedHmiRequest';
END_CASE

IF NOT HmiResponse.Accepted AND (HmiResponse.Diagnostic = '') THEN
    HmiResponse.Diagnostic := 'std.error.hmiRequestRejected';
ELSE
    HmiResponse.Diagnostic := HmiResponse.Diagnostic;
END_IF
_M_AuditHmiAccepted(Kind := HmiRequest.Kind, TargetPath := HmiRequest.TargetPath,
    Accepted := HmiResponse.Accepted);
HmiRequest.Secret := '';
HmiResponse.AckSequence := _hmiLastSequence;
END_METHOD

// §11.6 one owning projection helper; callers supply only event-specific fields.
METHOD PRIVATE _M_HostEvent : BOOL
VAR_INPUT
    Kind          : E_HostEventKind;
    PartUid       : STRING(64);
    Subject       : STRING(80);
    Value         : STRING(80);
    Verdict       : E_Verdict;
    ReasonCode    : E_Reason;
END_VAR
_M_HostEvent := HostEvents.Emit(Kind := Kind,
    StationPath := _name, PartUid := PartUid, Subject := Subject,
    Value := Value, Verdict := Verdict, ReasonCode := ReasonCode);
END_METHOD

// §3.4.1/§3.14.4 — default per-mode switch policy. Station config (§3.8a) may
// overwrite ModePolicy[] after this. By FRAMEWORK DEFAULT a mode change while a
// sequence runs performs an IMMEDIATE software abort (E-stop-like, not a safety
// function, §3.14.4) — so Style defaults to IMMEDIATE. GRACEFUL completion is an
// opt-in: a Unit overrides OnModeExit to stop-after-cycle, or station config sets
// Style := GRACEFUL for a mode. Shield only governs acceptance while running.
METHOD PROTECTED _M_InitModePolicy
VAR
    i : INT;
END_VAR
FOR i := 0 TO PL_Fraktal.MODE_COUNT-1 DO
    ModePolicy[i].Shield := E_ModeSwitchShield.CONFIRM;
    ModePolicy[i].Style  := E_ModeSwitchStyle.IMMEDIATE;
END_FOR
// Setup modes a running machine may not leave without an explicit Stop first.
ModePolicy[TO_INT(E_Mode.CHANGEOVER)].Shield := E_ModeSwitchShield.BLOCKED_WHILE_RUNNING;
ModePolicy[TO_INT(E_Mode.CALIBRATION)].Shield:= E_ModeSwitchShield.BLOCKED_WHILE_RUNNING;
// HOME and MANUAL are freely interruptible; both inherit the IMMEDIATE default.
ModePolicy[TO_INT(E_Mode.HOME)].Shield       := E_ModeSwitchShield.INTERRUPTIBLE;
ModePolicy[TO_INT(E_Mode.MANUAL)].Shield     := E_ModeSwitchShield.INTERRUPTIBLE;
END_METHOD

// §8.5.1 — pure recompute of A/P/Q/OEE from the accumulators (testable in isolation).
// Invalid factors are OMITTED from the product, never assumed 100% (O7).
METHOD PROTECTED _M_OeeCompute
VAR
    total : UDINT;
    denomA: UDINT;
END_VAR
denomA := Oee.RunMs + Oee.DownMs;
Oee.AvailValid := denomA > 0;
IF Oee.AvailValid THEN
    Oee.Availability := UDINT_TO_REAL(Oee.RunMs) / UDINT_TO_REAL(denomA);
ELSE
    Oee.Availability := 0.0;
END_IF
Oee.PerfValid := (Oee.IdealCycleMs > 0) AND (Oee.RunMs > 0);
IF Oee.PerfValid THEN
    Oee.Performance := UDINT_TO_REAL(Oee.IdealCycleMs) * UDINT_TO_REAL((GoodCount - _oeeGoodBase) + (NokCount - _oeeNokBase))
                       / UDINT_TO_REAL(Oee.RunMs);
    IF Oee.Performance > 1.0 THEN
        Oee.Performance := 1.0;          // faster than ideal caps at 100% (standard practice)
    END_IF
ELSE
    Oee.Performance := 0.0;
END_IF
total := (GoodCount - _oeeGoodBase) + (NokCount - _oeeNokBase);
Oee.QualValid := total > 0;
IF Oee.QualValid THEN
    Oee.Quality := UDINT_TO_REAL(GoodCount - _oeeGoodBase) / UDINT_TO_REAL(total);
ELSE
    Oee.Quality := 0.0;
END_IF
// product of VALID factors only; OEE valid iff at least one factor is valid
Oee.Oee := 1.0;
Oee.OeeValid := FALSE;
IF Oee.AvailValid THEN Oee.Oee := Oee.Oee * Oee.Availability; Oee.OeeValid := TRUE; END_IF
IF Oee.PerfValid  THEN Oee.Oee := Oee.Oee * Oee.Performance;  Oee.OeeValid := TRUE; END_IF
IF Oee.QualValid  THEN Oee.Oee := Oee.Oee * Oee.Quality;      Oee.OeeValid := TRUE; END_IF
IF NOT Oee.OeeValid THEN
    Oee.Oee := 0.0;
END_IF
END_METHOD

// §8.5.1 — attribute elapsed time to run/down/idle, recompute factors, sample ring.
METHOD PROTECTED _M_OeeUpdate
VAR
    currentTime : TIME;
    deltaMs     : UDINT;
END_VAR
currentTime := TIME();                 // monotonic duration clock
IF _oeeLast = T#0S THEN
    _oeeLast := currentTime;
    RETURN;
END_IF
deltaMs := TIME_TO_UDINT(currentTime) - TIME_TO_UDINT(_oeeLast); // wrap-safe on UDINT subtraction
_oeeLast := currentTime;
IF _exec = E_ExecState.BUSY THEN
    Oee.RunMs := Oee.RunMs + deltaMs;
ELSIF (_exec = E_ExecState.ERROR) OR AlarmLog.Blocking THEN
    Oee.DownMs := Oee.DownMs + deltaMs;
ELSE
    Oee.IdleMs := Oee.IdleMs + deltaMs;
END_IF
_M_OeeCompute();
_oeeSampMs := _oeeSampMs + deltaMs;
IF _oeeSampMs >= PL_Fraktal.OEE_SAMPLE_MS THEN
    _oeeSampMs := 0;
    OeeTrendHead := (OeeTrendHead MOD PL_Fraktal.MAX_OEE_SAMPLES) + 1;
    OeeTrend[OeeTrendHead].Availability := Oee.Availability;
    OeeTrend[OeeTrendHead].Performance  := Oee.Performance;
    OeeTrend[OeeTrendHead].Quality      := Oee.Quality;
    OeeTrend[OeeTrendHead].Oee          := Oee.Oee;
    OeeTrend[OeeTrendHead].OeeValid     := Oee.OeeValid;
END_IF
END_METHOD

// §3.16.3 EVENT_PART_PROCESSING_ABORTED — the part leaves without a valid result
// (fault, abort, manual removal). Called automatically on Unit ERROR entry.
METHOD PROTECTED _M_PartAborted
IF (_carrier = 0) OR NOT Part.Present THEN
    RETURN;
END_IF
Part.Result.Verdict := E_Verdict.NONE;
IF (_exec = E_ExecState.ERROR) AND (Part.Result.ReasonCode = E_Reason.NONE) THEN
    Part.Result.ReasonCode := _diag.ReasonCode;
END_IF
_M_PartEvent(Reason := E_Reason.EVENT_PART_PROCESSING_ABORTED,
    Text := 'std.event.partAborted: ');
_M_HostEvent(Kind := E_HostEventKind.PROCESSING_ABORTED, PartUid := Part.Uid,
    Subject := '', Value := '',
    Verdict := E_Verdict.NONE, ReasonCode := Part.Result.ReasonCode);
Part.Present := FALSE;
END_METHOD

// §3.16.3 — one canonical part-lifecycle event: instant come+gone MESSAGE ring entry.
METHOD PRIVATE _M_PartEvent
VAR_INPUT
    Reason : E_Reason;
    Text : STRING(255);
END_VAR
VAR
    slot : INT;
    txt : STRING(255);
END_VAR
txt := CONCAT(Text, Part.Uid);
slot := AlarmLog.Raise(Reason := Reason, Text := txt, Source := _name,
    Severity := E_Severity.LOW, Category := E_Category.PROCESS,
    ResetClass := E_ResetClass.AUTO_RESET);
IF slot > 0 THEN
    AlarmLog.Gone(Slot := slot);
END_IF
END_METHOD

// §3.16.3 EVENT_PART_PROCESSED — stamp the verdict, write the carrier FIRST
// (result-before-event contract), then raise the event. The Uid and result stay
// published until the next part so the HMI shows the last outcome.
METHOD PROTECTED _M_PartProcessed : BOOL
VAR_INPUT
    Verdict : E_Verdict;
    Reason : E_Reason;
END_VAR
_M_PartProcessed := FALSE;
IF (_carrier = 0) OR NOT Part.Present THEN
    RETURN;
END_IF
// A reject without a first-out reason cannot satisfy the KPI or host contract.
// Reject it before writing the carrier so result-before-event remains atomic.
IF (Verdict = E_Verdict.NOK) AND (Reason = E_Reason.NONE) THEN
    _M_Fault(E_Reason.RESULT_RECORD_REJECTED, 'std.error.nokReasonRequired');
    RETURN;
END_IF
Part.Result.Verdict := Verdict;
Part.Result.ReasonCode := Reason;
Part.Result.StationPath := _name;
Part.Result.Stamp := F_Now();
Part.Result.TimeSynchronized := F_TimeSynchronized();
IF NOT _carrier.WriteResult(Ctx := Part) THEN
    _M_Fault(E_Reason.CARRIER_WRITE_FAILED, 'std.error.partCarrierWriteFailed');
    RETURN;
END_IF
// §8.11.2 — counters increment HERE, from the verdict; an NOK carries its
// first-out ReasonCode so scrap is analysable by cause (§8.8 vocabulary).
CASE Verdict OF
    E_Verdict.OK:     CountGood();
    E_Verdict.NOK:
        IF NOT CountNok(Reason := Reason) THEN
            RETURN;
        END_IF
    E_Verdict.REWORK: CountRework();
ELSE
    ;                                // NONE: no count — the part left unjudged
END_CASE
_M_PartEvent(Reason := E_Reason.EVENT_PART_PROCESSED, Text := 'std.event.partProcessed: ');
_M_HostEvent(Kind := E_HostEventKind.PROCESSED, PartUid := Part.Uid,
    Subject := '', Value := '',
    Verdict := Verdict, ReasonCode := Reason);
Part.Present := FALSE;
_M_PartProcessed := TRUE;
END_METHOD

// §3.16.3 EVENT_PART_RECEIVED — confirm identity at station entry via the carrier.
// FALSE with a CARRIER_READ_FAILED fault on a failed read (never silent), FALSE
// silently when no carrier is configured (§3.9 feature selectability).
METHOD PROTECTED _M_PartReceived : BOOL
VAR
    i : INT;
END_VAR
_M_PartReceived := FALSE;
IF _carrier = 0 THEN
    RETURN;
END_IF
Part.Uid := '';                              // station entry = fresh identity read
IF NOT _carrier.ReadContext(Ctx := Part) THEN
    _M_Fault(E_Reason.CARRIER_READ_FAILED, 'std.error.partCarrierReadFailed');
    RETURN;
END_IF
Part.Result.Verdict := E_Verdict.NONE;       // this station's outcome starts empty
Part.Result.ReasonCode := E_Reason.NONE;
Part.Result.StationPath := _name;
FOR i := 1 TO PL_Fraktal.MAX_RESULTS DO
    Part.Result.Records[i].Name := '';
END_FOR
_M_PartEvent(Reason := E_Reason.EVENT_PART_RECEIVED, Text := 'std.event.partReceived: ');
_M_HostEvent(Kind := E_HostEventKind.PART_RECEIVED, PartUid := Part.Uid,
    Subject := '', Value := '',
    Verdict := E_Verdict.NONE, ReasonCode := E_Reason.NONE);
_M_PartReceived := TRUE;
END_METHOD

// §3.16.1 — append one measured value to this part's result (test cells).
// FALSE when the bounded record table is full (RESULT_RECORD_REJECTED semantics).
METHOD PROTECTED _M_PartRecord : BOOL
VAR_INPUT
    RecordName : STRING(64);
    Value : LREAL;
    Minimum : LREAL;
    Maximum : LREAL;
    Target : LREAL;
    EngUnit : STRING(16);
END_VAR
VAR
    i : INT;
END_VAR
_M_PartRecord := FALSE;
IF NOT Part.Present THEN
    RETURN;
END_IF
FOR i := 1 TO PL_Fraktal.MAX_RESULTS DO
    IF Part.Result.Records[i].Name = '' THEN
        Part.Result.Records[i].Name := RecordName;
        Part.Result.Records[i].Value := Value;
        Part.Result.Records[i].Minimum := Minimum;
        Part.Result.Records[i].Maximum := Maximum;
        Part.Result.Records[i].Target := Target;
        Part.Result.Records[i].Unit := EngUnit;
        Part.Result.Records[i].InTol := (Maximum <= Minimum)
            OR ((Value >= Minimum) AND (Value <= Maximum));
        _M_PartRecord := TRUE;
        RETURN;
    END_IF
END_FOR
END_METHOD

// §3.16.3 EVENT_PART_PROCESSING_STARTED — the value-adding sequence begins.
METHOD PROTECTED _M_PartStarted
IF (_carrier = 0) OR NOT Part.Present THEN
    RETURN;
END_IF
_M_PartEvent(Reason := E_Reason.EVENT_PART_PROCESSING_STARTED,
    Text := 'std.event.partProcessingStarted: ');
_M_HostEvent(Kind := E_HostEventKind.PROCESSING_STARTED, PartUid := Part.Uid,
    Subject := '', Value := '',
    Verdict := E_Verdict.NONE, ReasonCode := E_Reason.NONE);
END_METHOD

